# B&R Automation Studio project ProjectOrionBms (part 2)

#### AMS_Receive.st
```iecst
ACTION AMS_Receive:
	// Timer used for disconnection detection of AMS
	TON_amsDisconnected.PT   := T#200ms;	// Set timeout period
	TON_amsDisconnected.IN 	 := TRUE;		// Enable timer

	// Timer used for disconnection detection of shunt
	TON_shuntDisconnected.PT := T#200ms; 	// Set timeout period
	TON_shuntDisconnected.IN := TRUE;		// Enable timer

	FOR i := 0 TO 10 DO
		ArCanReceive_0(); // Run function block => Get next data frame

		(* If a new message has been received *)
		IF ArCanReceive_0.NewDataValid THEN
			messageCounterRec := messageCounterRec + 1;
			// Figure out if it is a shunt message
			IF ArCanReceive_0.ReceivedFrame.ID > SHUNT_ID_BASE AND ArCanReceive_0.ReceivedFrame.ID < (SHUNT_ID_BASE+16#30) THEN
				// Its a shunt message
				frameId := ArCanReceive_0.ReceivedFrame.ID - SHUNT_ID_BASE;
				// Look up message decoding
				CASE frameId OF
					16#021: msg_shunt_021;
					16#022: msg_shunt_022;
					16#023: msg_shunt_023;
//					16#025: msg_shunt_025;
					16#026: msg_shunt_026;
					16#027: msg_shunt_027;
					16#028: msg_shunt_028;
					ELSE (* Message not registered in system *)
				END_CASE

				(* Reset timer for disconnection detection *)
				TON_shuntDisconnected.IN := FALSE;

			// Figure out if the message is a ORION Message
			ELSIF ArCanReceive_0.ReceivedFrame.ID >= RX_ORION_ID_BASE AND ArCanReceive_0.ReceivedFrame.ID < (RX_ORION_ID_BASE+16#30) THEN
				// It is an ORION messagemm
				frameId := ArCanReceive_0.ReceivedFrame.ID - RX_ORION_ID_BASE;

				// Look up message decoding
				CASE frameId OF
					//16#000: msg_orion_000;
					16#001: msg_orion_001;
					16#002: msg_orion_002;
					16#003: msg_orion_003;
					16#004: msg_orion_004;
					16#010: msg_orion_010;
					16#011: msg_orion_011;

					ELSE // Not a message in the system
				END_CASE

			ELSE
				// Its an AMS message
				frameId := UDINT_TO_UINT(ArCanReceive_0.ReceivedFrame.ID) - RX_CAN_ID_BASE;

				// Look up message decoding
				CASE frameId OF
					16#000: msg_ams_000;
					16#011: msg_ams_011;
					16#012: msg_ams_012;
					16#013: msg_ams_013;
					16#014: msg_ams_014;
					ELSE (* Message not registered in system *)
				END_CASE

				TON_amsDisconnected.IN := FALSE; // Reset Timer
			END_IF;
		ELSE
			EXIT;
		END_IF
	END_FOR;

	(* If timeout occurres on AMS timer set AMS disconnect status flag *)
	TON_amsDisconnected();
	gAMS.status.disconnected := TON_amsDisconnected.Q;

	(* If timeout occurres on shunt timer set shunt disconnect status flag *)
	TON_shuntDisconnected();
	gShunt.status.disconnected := TON_shuntDisconnected.Q;

END_ACTION
```

### Program Logical/Dashboard/Dashboard

#### ErrorDashboard.st
```iecst
ACTION ErrorDashboard:

	gDashboard.outputs.com_error_Datalog 				:= NOT gDataLogging.status.dataloggingActive; // Datalogging not active
	gDashboard.outputs.com_error_SC 					:= NOT gSafetyChain.status.scOK_notEnabled; // Safety chain not ok
	gDashboard.outputs.com_error_Shunt 					:= NOT gShunt.status.ok; // Shunt error
	gDashboard.outputs.com_error_AMS 					:= NOT gAMS.status.ok; // AMS error
	gDashboard.outputs.com_error_Dashboard 				:= NOT gDashboard.status.ok; // Dashboard error
	gDashboard.outputs.com_error_3rd_Inv 				:= NOT gInverters.inverter[3].status.ok; // 3rd inverter error
	gDashboard.outputs.com_error_2nd_Inv 				:= NOT gInverters.inverter[2].status.ok; // 2nd inverter error
	gDashboard.outputs.com_error_1st_Inv 				:= NOT gInverters.inverter[1].status.ok; // 1st inverter error
	gDashboard.outputs.com_error_0_Inv 					:= NOT gInverters.inverter[0].status.ok; // [0] inverter error
	gDashboard.outputs.com_error_INS 					:= NOT gINS.status.ok; // INS error
	gDashboard.outputs.com_error_SteeringAngle 			:= gSteeringAngle.status.errorOutOfRange; // Steering angle out of range
	gDashboard.outputs.com_error_BreakPressure_Front 	:= gBraking.status.errorOutOfRangeFront; // Brake Pressure out-of-range (Front)
	gDashboard.outputs.com_error_BreakPressure_Back 	:= gBraking.status.errorOutOfRangeRear; // Brake Pressure out-of-range (Rear)
	gDashboard.outputs.com_error_TorquePedal 			:= gTorqueSensor.status.criticalError; // One of the Torque Pedal sensors out of range
	gDashboard.outputs.com_error_TorquePedal_Plausi 	:= gTorqueSensor.status.plausibilityError; // Plausibility error on Torque pedal
	gDashboard.outputs.com_error_RTDS 					:= NOT gRTDS.status.ok; // RTDS error
	gDashboard.outputs.com_error_Cooling	 			:= NOT gCooling.status.ok; // Cooling error
	gDashboard.outputs.com_error_LV 					:= gLowVoltageBattery.status.empty; // Low Voltage Battery critically low
	gDashboard.outputs.com_error_HighTemperature 		:= gCooling.status.warningHighTemperature;
END_ACTION
```

#### errors.st
```iecst
ACTION errors:
	// Change this variable to indicate what error is active in the system.
	// 0 = No error
	gDashboard.status.errorCode := 0;
END_ACTION
```

#### Main.st
```iecst
PROGRAM _INIT
	(* Device *)
	deviceName 						:= 'IF6.ST1.IF1';
	(* Bus *)
	ArCanSetBaudrate_0.Baudrate 	:= 1000000;
	(* Tramsit *)
	ArCanSend_0.Frame.Format 		:= arCAN_11BIT;
	(* Receive *)
	ArCanReceive_0.Format 			:= arCAN_11BIT;
	ArCanReceive_0.QueueSize		:= 100;
	ArCanReceive_0.IDMask			:= arCAN_RECEIVE_ALL;

	communicationState 				:= S_INIT;

	scLedState 						:= OFF;
	ledLVState 						:= 0;

	RX_CAN_ID_BASE 					:= 16#580;
	TX_CAN_ID_BASE 					:= 16#580;

END_PROGRAM

PROGRAM _CYCLIC

	(* Determine of the Dashboard has an error or is working properly*)
	gDashboard.status.ok := NOT gDashboard.status.DashboardDisconnected AND gDashboard.status.errorCode = 0;

	(* LED Control *)
	ledAMS;
	ledDV;
	ledEBS;
	ledIMD;
	ledLV;
	ledREADY;
	ledSC;
	ledTS_OFF;
	ErrorDashboard;

	(* Send and receive messages *)
	can;

	(* Error *)
	errors;

	// Log button presses
	IF EDGEPOS(gDashboard.inputs.di_button1) THEN
		gEventLog.newEventString := 'Button 1 pressed';
		logEvent;
	END_IF;
	IF EDGEPOS(gDashboard.inputs.di_button2) THEN
		gEventLog.newEventString := 'Button 2 pressed';
		logEvent;
	END_IF;
	IF EDGEPOS(gDashboard.inputs.di_button3) THEN
		gEventLog.newEventString := 'Button 3 pressed';
		logEvent;
	END_IF;
	IF EDGEPOS(gDashboard.inputs.di_button4) THEN
		gEventLog.newEventString := 'Button 4 pressed';
		logEvent;
	END_IF;
	IF EDGEPOS(gDashboard.inputs.di_buttonSafety) THEN
		gEventLog.newEventString := 'Button Safety pressed';
		logEvent;
	END_IF;
	IF EDGEPOS(gDashboard.inputs.di_buttonTractive) THEN
		gEventLog.newEventString := 'Button Tractive pressed';
		logEvent;
	END_IF;
	IF EDGEPOS(gDashboard.inputs.di_buttonDrive) THEN
		gEventLog.newEventString := 'Button Drive pressed';
		logEvent;
	END_IF;

END_PROGRAM

PROGRAM _EXIT

END_PROGRAM
```

#### ledTS_OFF.st
```iecst
(* Control the TS_OFF LED *)
ACTION ledTS_OFF:
	IF gStateMachine.status.state = STATE_INITIALIZE THEN
		gDashboard.outputs.do_ledTS_OFF := TRUE;
	ELSE
		gDashboard.outputs.do_ledTS_OFF := NOT (gStateMachine.status.state = STATE_TRACTIVE OR  gStateMachine.status.state = STATE_DRIVE);
	END_IF;

END_ACTION
```

#### Program Logical/Dashboard/Dashboard/Receive

##### Receive_Bus.st
```iecst
ACTION Receive_Bus:

	TON_disconnectTimer.PT := T#200ms;
	TON_disconnectTimer.IN := TRUE;

	FOR i := 0 TO UDINT_TO_USINT(LIMIT(0,ArCanReceive_0.QueueSize,255)) DO
		ArCanReceive_0(); // Run function block => Get next data frame
		(* If a new message has been received *)
		IF ArCanReceive_0.NewDataValid THEN
			(* Find which message is was and decode it *)

			frameIdOffset := ArCanReceive_0.ReceivedFrame.ID - RX_CAN_ID_BASE;
			CASE frameIdOffset OF
				16#050: msg_0x050;
				16#051: msg_0x051;
				16#052: msg_0x052;
				ELSE
				(* Message not registered in system *)
				gDashboard.status.unknownMessageReceived 	:= TRUE;
				gDashboard.status.unknownMessageID	 		:= ArCanReceive_0.ReceivedFrame.ID;
			END_CASE

			(* Enable timer to check if dashboard is disconnected *)
			TON_disconnectTimer.IN := FALSE;
			gDashboard.status.DashboardDisconnected := FALSE;
		ELSE
			EXIT;
		END_IF
	END_FOR;

	TON_disconnectTimer();

	(* If 200 ms is passed without message, set dashboard disconnect status flag *)
	IF TON_disconnectTimer.Q = TRUE THEN
		gDashboard.status.DashboardDisconnected := TRUE;
	END_IF

	gDashboard.status.canFramesLost := ArCanReceive_0.NumberOfLostFrames <> 0;

END_ACTION
```

### globalBraking.typ
```iecst
TYPE
	gBraking_cmd_typ : 	STRUCT
		brakePressureFront : INT;
		brakePressureRear : INT;
	END_STRUCT;
	gBraking_typ : 	STRUCT
		status : gBraking_status_typ;
		inputs : gBraking_inputs_typ;
		outputs : gBraking_outputs_typ;
		data : gBraking_data_typ;
		cmd : gBraking_cmd_typ;
	END_STRUCT;
	gBraking_status_typ : 	STRUCT
		ok : BOOL;
		errorOutOfRangeFront : BOOL;
		errorOutOfRangeRear : BOOL;
		softBraking : BOOL;
		hardBraking : BOOL;
	END_STRUCT;
	gBraking_inputs_typ : 	STRUCT
		ai_brakePressureFront : INT;
		ai_brakePressureRear : INT;
	END_STRUCT;
	gBraking_outputs_typ : 	STRUCT
		do_brakeLight : BOOL;
	END_STRUCT;
	gBraking_data_typ : 	STRUCT
		pressurePercentageFront : REAL;
		pressurePercentageRear : REAL;
		pressurePercentage : REAL;
		pressureBarRear : REAL;
		pressureBarFront : REAL;
	END_STRUCT;
END_TYPE
```

### globalBraking.var
```iecst
VAR
	gSoftBrakingForced : BOOL;
	gBraking : gBraking_typ;
END_VAR
```

### globalTorqueSensor.var
```iecst
VAR
	gTorqueSensor : gTorqueSensor_typ;
END_VAR
```

### Program Logical/Sensors/Sensors (IEC)

#### Main.st - Init, cyclic, exit code
```iecst
PROGRAM _INIT
	(* Initialize all the sensors *)
	// Accelerometer
	AccelerometerInit;

	// Braking Pedal Sensor
	BrakingPedalInit;

	// Torque Pedal Sensor
	TorquePedalInit;

	// Steering Angle Sensor
	SteeringAngleInit;

	// Low voltage battery
	LowVoltageBatteryInit;

	// Suspension Measurement
	SuspensionMeasInit;
END_PROGRAM

PROGRAM _CYCLIC
	//Accelerometer
	Accelerometer;

	// Handle Braking Pedal Sensor
	BrakingPedal;

	// Handle TorquePedal Sensor
	TorquePedal;

	// Handle Braking Pedal Sensor
	SteeringAngle;

	// Low voltage battery
	LowVoltageBattery;

	// Suspension Measurement
	SuspensionMeas;
END_PROGRAM

PROGRAM _EXIT
	(* Insert code here *)

END_PROGRAM
```

#### Types.typ - Local data types
```iecst
TYPE
	accelerometer_constants_typ : 	STRUCT
		VOLTAGE_MIN : UDINT;
		VOLTAGE_MAX : UDINT;
		MEASUREMENT_RES : UDINT;
		SENSOR_SUPPLY_VOLTAGE : UDINT;
		SENSITIVITY : REAL;
		ZERO_POINT : REAL;
	END_STRUCT;
	accelerometer_input_typ : 	STRUCT
		x_direction : INT;
		y_direction : INT;
		z_direction : INT;
	END_STRUCT;
	accelerometer_status_typ : 	STRUCT
		voltage_x : REAL;
		voltage_y : REAL;
		voltage_z : REAL;
		acceleration_x : REAL;
		acceleration_y : REAL;
		acceleration_z : REAL;
	END_STRUCT;
	accelerometer_typ : 	STRUCT
		constants : accelerometer_constants_typ;
		input : accelerometer_input_typ;
		status : accelerometer_status_typ;
	END_STRUCT;
	braking_pedal_constants_typ : 	STRUCT
		frontWarningLimitMaxMax : UINT;
		frontWarningLimitMax : UINT;
		frontWarningLimitMin : UINT;
		frontWarningLimitMinMin : UINT;
		rearWarningLimitMaxMax : UINT;
		rearWarningLimitMax : UINT;
		rearWarningLimitMin : UINT;
		rearWarningLimitMinMin : UINT;
		softBrakingLimit : UINT;
		hardBrakingLimit : UINT;
	END_STRUCT;
	braking_pedal_variables_typ : 	STRUCT
		brakingPedalFrontMax : UINT;
		brakingPedalFrontMin : UINT;
		brakingPedalRearMax : UINT;
		brakingPedalRearMin : UINT;
		slope : REAL;
	END_STRUCT;
	lv_battery_constants_typ : 	STRUCT
		HighLimit : REAL;
		LowLimit : REAL;
	END_STRUCT;
	lv_battery_variable_typ : 	STRUCT
		TON_batteryEmpty : TON;
		TON_batteryFull : TON;
	END_STRUCT;
	steering_angle_constants_typ : 	STRUCT
		highLimit : UINT;
		lowLimit : UINT;
		disconnectionLimit : UINT;
		MAX_ANGLE : REAL;
		MIN_ANGLE : REAL;
	END_STRUCT;
	steering_angle_variables_typ : 	STRUCT
		steeringWheelAngleStr : STRING[80];
		wheelAngleStr : STRING[80];
		leftValue : UINT;
		rightValue : UINT;
	END_STRUCT;
	suspension_const_typ : 	STRUCT
		VOLTAGE_MIN : UDINT;
		VOLTAGE_MAX : UDINT;
		MEASUREMENT_RES : UDINT;
		SENSOR_SUPPLY_VOLTAGE : UDINT;
		TRAVEL_RES : UDINT;
	END_STRUCT;
	suspension_input_typ : 	STRUCT
		linearPosSensor : ARRAY[0..3]OF INT;
	END_STRUCT;
	suspension_status_typ : 	STRUCT
		travelRR : REAL;
		travelFR : REAL;
		travelRL : REAL;
		travelFL : REAL;
		voltageRR : REAL;
		voltageFR : REAL;
		voltageRL : REAL;
		voltageFL : REAL;
	END_STRUCT;
	suspension_typ : 	STRUCT
		constants : suspension_const_typ;
		input : suspension_input_typ;
		status : suspension_status_typ;
	END_STRUCT;
	torque_pedal_constants_typ : 	STRUCT
		lowLimit2 : UINT;
		highLimit2 : UINT;
		lowLimit1 : UINT;
		highLimit1 : UINT;
		torqueOffUpperHysteresis : REAL;
		torqueOffLowerHysteresis : REAL;
	END_STRUCT;
	torque_pedal_variables_typ : 	STRUCT
		torquePedalMax2 : UINT;
		torquePedalMax1 : UINT;
		torquePedalMin2 : UINT;
		torquePedalMin1 : UINT;
		TON_torqueOff : TON;
		slope : REAL;
	END_STRUCT;
END_TYPE
```

#### Variables.var - Local variables
```iecst
VAR
	accelerometer : accelerometer_typ;
	brakingPedalVariables : braking_pedal_variables_typ;
	brakingPedalConstants : braking_pedal_constants_typ;
	torquePedalConstants : torque_pedal_constants_typ;
	torquePedalVariables : torque_pedal_variables_typ;
	steeringAngleConstants : steering_angle_constants_typ;
	steeringAngleVariables : steering_angle_variables_typ;
	lvBatteryConstants : lv_battery_constants_typ;
	lvBatteryVariables : lv_battery_variable_typ;
END_VAR
VAR RETAIN
	maxTorquePercentThrottle : USINT;
END_VAR
VAR
	suspension : suspension_typ;
END_VAR
```

#### BrakingPedal.st
```iecst
ACTION BrakingPedalInit:
	(* Sensor limit values *)
	brakingPedalVariables.brakingPedalRearMax 		:= 8000;
	brakingPedalVariables.brakingPedalRearMin 		:= 1655;
	brakingPedalVariables.brakingPedalFrontMax 		:= 8000;
	brakingPedalVariables.brakingPedalFrontMin 		:= 1655;

	(* Braking limits *)
	brakingPedalConstants.hardBrakingLimit			:= 5400;
	brakingPedalConstants.softBrakingLimit			:= 2200;

	(* Upper limit symboling an electrical fault *)
//	brakingPedalConstants.frontWarningLimitMaxMax 	:= brakingPedalVariables.brakingPedalFrontMax + 500;
//	brakingPedalConstants.rearWarningLimitMaxMax 	:= brakingPedalVariables.brakingPedalRearMax  + 500;
	brakingPedalConstants.frontWarningLimitMaxMax 	:= 15250;
	brakingPedalConstants.rearWarningLimitMaxMax 	:= 15250;

	(* Upper limit symboling a mechanical fault *)
	brakingPedalConstants.frontWarningLimitMax 		:= brakingPedalVariables.brakingPedalFrontMax + 100;
	brakingPedalConstants.rearWarningLimitMax 		:= brakingPedalVariables.brakingPedalRearMax  + 100;

	(* Lower limit symboling a mechanical fault *)
	brakingPedalConstants.frontWarningLimitMin 		:= brakingPedalVariables.brakingPedalFrontMin - 100;
	brakingPedalConstants.rearWarningLimitMin 		:= brakingPedalVariables.brakingPedalRearMin  - 100;

	(* Lower limit symboling an electrical fault *)
	brakingPedalConstants.frontWarningLimitMinMin 	:= brakingPedalVariables.brakingPedalFrontMin - 500;
	brakingPedalConstants.rearWarningLimitMinMin 	:= brakingPedalVariables.brakingPedalRearMin  - 500;

END_ACTION

ACTION BrakingPedal:
	(* Detect if brake pedal is being pressed lightly *)
	gBraking.status.softBraking 		 := INT_TO_UINT(gBraking.inputs.ai_brakePressureRear)  > brakingPedalConstants.softBrakingLimit OR
											gSoftBrakingForced;

	(* Detect hard braking *)
	gBraking.status.hardBraking 		 := INT_TO_UINT(gBraking.inputs.ai_brakePressureFront) > brakingPedalConstants.hardBrakingLimit OR
										    INT_TO_UINT(gBraking.inputs.ai_brakePressureRear)  > brakingPedalConstants.hardBrakingLimit;

	(* Control brakelight *)
	IF gStateMachine.status.state <> STATE_INITIALIZE THEN
		gBraking.outputs.do_brakeLight   := gBraking.status.softBraking;
	END_IF

	(* Check if brake pressures are out of range *)
	// If brake pressure front get above limit, an error message is shown.
	gBraking.status.errorOutOfRangeFront := INT_TO_UINT(gBraking.inputs.ai_brakePressureFront) >= brakingPedalConstants.frontWarningLimitMax OR
											INT_TO_UINT(gBraking.inputs.ai_brakePressureFront) <= brakingPedalConstants.frontWarningLimitMin;

	// If brake pressure rear get above limit, an error message is shown.
	gBraking.status.errorOutOfRangeRear := 	INT_TO_UINT(gBraking.inputs.ai_brakePressureRear) >= brakingPedalConstants.rearWarningLimitMax OR
											INT_TO_UINT(gBraking.inputs.ai_brakePressureRear) <= brakingPedalConstants.rearWarningLimitMin;

	(* Calculate pedal percentages *)
	IF NOT gBraking.status.errorOutOfRangeFront THEN
		brakingPedalVariables.slope := (100.00)/(UINT_TO_REAL(brakingPedalVariables.brakingPedalFrontMax) - UINT_TO_REAL(brakingPedalVariables.brakingPedalFrontMin));
		gBraking.data.pressurePercentageFront := LIMIT(0 ,brakingPedalVariables.slope * (INT_TO_REAL(gBraking.inputs.ai_brakePressureFront)-UINT_TO_REAL(brakingPedalVariables.brakingPedalFrontMin)),100);
	ELSE
		gBraking.data.pressurePercentageFront := 0;
	END_IF;

	IF NOT gBraking.status.errorOutOfRangeRear THEN
		brakingPedalVariables.slope := (100.00)/(UINT_TO_REAL(brakingPedalVariables.brakingPedalRearMax) - UINT_TO_REAL(brakingPedalVariables.brakingPedalRearMin));
		gBraking.data.pressurePercentageRear := LIMIT(0 ,brakingPedalVariables.slope * (INT_TO_REAL(gBraking.inputs.ai_brakePressureRear)-UINT_TO_REAL(brakingPedalVariables.brakingPedalRearMin)),100);
	ELSE
		gBraking.data.pressurePercentageRear := 0;
	END_IF;

	gBraking.data.pressurePercentage := (gBraking.data.pressurePercentageFront + gBraking.data.pressurePercentageRear)/2.0;

	(* Determine if the brake pedal + sensors are working properly *)
	gBraking.status.ok := NOT gBraking.status.errorOutOfRangeFront AND NOT gBraking.status.errorOutOfRangeRear;

	// Calculate actual pressure
	gBraking.data.pressureBarFront 	:= ((INT_TO_REAL(gBraking.inputs.ai_brakePressureFront)*10/32768)-0.5)*40;
	gBraking.data.pressureBarRear	:= ((INT_TO_REAL(gBraking.inputs.ai_brakePressureRear)*10/32768)-0.5)*40;

END_ACTION
```

#### TorquePedal.st
```iecst
ACTION TorquePedalInit:
	(* Sensor edge values *)
	torquePedalVariables.torquePedalMin1 	:= 13636;
	torquePedalVariables.torquePedalMin2 	:= 2415;
	torquePedalVariables.torquePedalMax1 	:= 21181;
	torquePedalVariables.torquePedalMax2 	:= 7947;

	// Constant for limit torque percent
	IF maxTorquePercentThrottle = 0 THEN
		maxTorquePercentThrottle := 50; // Change to 100 for max torque, 50 is a bit over nominal  torque. Max= 21NM, Nominal = 9,8Nm
	END_IF;
	gTorqueSensor.status.maxTorquePercent := maxTorquePercentThrottle;

	(* Range for torque sensor 1 *)
	torquePedalConstants.highLimit1 := torquePedalVariables.torquePedalMax1 + 200;
	torquePedalConstants.lowLimit1  := 0;

	(* Range for torque sensor 2 *)
	torquePedalConstants.highLimit2 := torquePedalVariables.torquePedalMax2 + 200;
	torquePedalConstants.lowLimit2 	:= 0;

	(* Torque off hysteresis values *)
	torquePedalConstants.torqueOffUpperHysteresis := 25; // [%]
	torquePedalConstants.torqueOffLowerHysteresis := 5;  // [%]

	(* Plausibility check disable (for test setup) *)
	gTorqueSensor.cmd.disablePlausibilityCheck := FALSE;
END_ACTION

ACTION TorquePedal:
	// Percent of MAX torque at full throttle:
	gTorqueSensor.status.maxTorquePercent := maxTorquePercentThrottle;

	gTorqueSensor.status.errorOutOfRangeSensor1 := 	INT_TO_UINT(gTorqueSensor.inputs.torque1) > torquePedalConstants.highLimit1 OR
													INT_TO_UINT(gTorqueSensor.inputs.torque1) < torquePedalConstants.lowLimit1;

	gTorqueSensor.status.errorOutOfRangeSensor2 := 	INT_TO_UINT(gTorqueSensor.inputs.torque2) > torquePedalConstants.highLimit2 OR
													INT_TO_UINT(gTorqueSensor.inputs.torque2) < torquePedalConstants.lowLimit2;

	(* Calculate pedal percentages *)

	// Sensor 1
	IF NOT gTorqueSensor.status.errorOutOfRangeSensor1 THEN
		torquePedalVariables.slope := (100)/(UINT_TO_REAL(torquePedalVariables.torquePedalMax1) - UINT_TO_REAL(torquePedalVariables.torquePedalMin1));
		gTorqueSensor.data.torque1Percent := LIMIT(0 ,torquePedalVariables.slope * (INT_TO_REAL(gTorqueSensor.inputs.torque1)-(10+UINT_TO_REAL(torquePedalVariables.torquePedalMin1))),100);
	ELSE
		gTorqueSensor.data.torque1Percent := 0;
	END_IF;
	// gTorqueSensor.status.maxTorquePercent TODO: USE THIS FOR SCALING
	// Sensor 2
	IF NOT gTorqueSensor.status.errorOutOfRangeSensor2 THEN
		torquePedalVariables.slope := (100)/(UINT_TO_REAL(torquePedalVariables.torquePedalMax2) - UINT_TO_REAL(torquePedalVariables.torquePedalMin2));
		gTorqueSensor.data.torque2Percent := LIMIT(0 ,torquePedalVariables.slope * (INT_TO_REAL(gTorqueSensor.inputs.torque2)-UINT_TO_REAL(torquePedalVariables.torquePedalMin2)),100);
	ELSE
		gTorqueSensor.data.torque2Percent := 0;
	END_IF;

	// Sensor 1 is arbitrarily taken to be the torque percentage
	// Value is then scaled by desired power
	gTorqueSensor.status.torquePercentage := gTorqueSensor.data.torque1Percent*gTorqueSensor.status.maxTorquePercent/100;

	(* Test if torque sensor values are out of range of each other*)
	TorqueSensorsOutOfRange;
	TorqueOff;

	(* Report critical error if either of the torque pedal sensors leave their working range *)
	gTorqueSensor.status.criticalError := gTorqueSensor.status.errorOutOfRangeSensor1 OR gTorqueSensor.status.errorOutOfRangeSensor2 OR gTorqueSensor.status.plausibilityError;

	(* Determine if the torque pedal is working properly *)
	gTorqueSensor.status.ok := NOT gTorqueSensor.status.criticalError;

END_ACTION

(* Test if torque pedals are more than 10% different than each other *)
ACTION TorqueSensorsOutOfRange:
	IF gTorqueSensor.cmd.disablePlausibilityCheck THEN
		gTorqueSensor.status.plausibilityError := FALSE;
	ELSE
		// check if torque sensor 1 and 2 vary more than 5 %
		gTorqueSensor.status.plausibilityError := ABS(gTorqueSensor.data.torque1Percent - gTorqueSensor.data.torque2Percent) > 5;
	END_IF;
END_ACTION

ACTION TorqueOff:
	IF gTorqueSensor.status.torqueEnabled THEN
		(* Test the criterias for turning off the torque. If they are met start timer *)
		IF 	gBraking.status.softBraking AND
			(gTorqueSensor.data.torque1Percent >= torquePedalConstants.torqueOffUpperHysteresis OR
			 gTorqueSensor.data.torque2Percent >= torquePedalConstants.torqueOffUpperHysteresis OR
		 	 gORION.data.packPower >= 5.0) THEN

			torquePedalVariables.TON_torqueOff.PT := T#250ms;	// Set timer duration TODO: Change to 500 that is the limit in the rules
			torquePedalVariables.TON_torqueOff.IN := TRUE;		// Start timer
		ELSE
			torquePedalVariables.TON_torqueOff.IN := FALSE;		// Else stop timer
		END_IF

		IF torquePedalVariables.TON_torqueOff.Q THEN			// If timer runs out
			gTorqueSensor.status.torqueEnabled := FALSE;		// Remove torque
		ELSE
			gTorqueSensor.status.torqueEnabled := TRUE;			// Else keep torque
		END_IF;
	ELSE
		(* Test the criterias for turning on the torque *)
		gTorqueSensor.status.torqueEnabled := 	gTorqueSensor.data.torque1Percent < torquePedalConstants.torqueOffLowerHysteresis AND
												gTorqueSensor.data.torque2Percent < torquePedalConstants.torqueOffLowerHysteresis AND (NOT gBraking.status.softBraking);
		torquePedalVariables.TON_torqueOff.IN := FALSE;			// Make sure the torque timer is stopped
	END_IF
	torquePedalVariables.TON_torqueOff();						// Run torque timer
END_ACTION
```

#### SteeringAngle.st
```iecst
ACTION SteeringAngleInit:
	(* Sensor limit values *)
	steeringAngleVariables.leftValue 	:= 7460;
	steeringAngleVariables.rightValue 	:= 25580;

	(* Error detection values *)
	steeringAngleConstants.disconnectionLimit := 300;
	steeringAngleConstants.lowLimit 	:= steeringAngleVariables.leftValue  - 500;
	steeringAngleConstants.highLimit 	:= steeringAngleVariables.rightValue + 500;

	steeringAngleConstants.MAX_ANGLE 	:=  100.00;
	steeringAngleConstants.MIN_ANGLE 	:= -100.00;
END_ACTION

ACTION SteeringAngle:
	(* 	Check if sensor input is within working range
		If not report an error  	*)
	gSteeringAngle.status.disconnected := INT_TO_UINT(gSteeringAngle.inputs.angleSensor) < steeringAngleConstants.disconnectionLimit;
	gSteeringAngle.status.errorOutOfRange := (NOT gSteeringAngle.status.disconnected) AND (INT_TO_UINT(gSteeringAngle.inputs.angleSensor) > steeringAngleConstants.highLimit OR INT_TO_UINT(gSteeringAngle.inputs.angleSensor) < steeringAngleConstants.lowLimit);
	(* Summerize errors *)
	gSteeringAngle.status.error := gSteeringAngle.status.disconnected OR gSteeringAngle.status.errorOutOfRange;

	(* Calculate steering angle *)
	IF NOT gSteeringAngle.status.error THEN
		// No error
		IF INT_TO_UINT(gSteeringAngle.inputs.angleSensor) < steeringAngleVariables.leftValue THEN
			gSteeringAngle.data.angleDegrees := steeringAngleConstants.MAX_ANGLE;
		ELSIF INT_TO_UINT(gSteeringAngle.inputs.angleSensor) > steeringAngleVariables.rightValue THEN
			gSteeringAngle.data.angleDegrees := steeringAngleConstants.MIN_ANGLE;
		ELSE
			gSteeringAngle.data.angleDegrees := LIMIT(-100, (INT_TO_REAL(gSteeringAngle.inputs.angleSensor) - UINT_TO_REAL(steeringAngleVariables.leftValue))/(UINT_TO_REAL(steeringAngleVariables.rightValue) - UINT_TO_REAL(steeringAngleVariables.leftValue)) *
			(ABS(steeringAngleConstants.MAX_ANGLE) + ABS(steeringAngleConstants.MIN_ANGLE)) + steeringAngleConstants.MIN_ANGLE, 100)*(-1);
		END_IF;
	ELSE
		// Error
		gSteeringAngle.data.angleDegrees := 0;
	END_IF

	(* Determine if the steering angle sensor is working properly *)
	gSteeringAngle.status.ok := NOT gSteeringAngle.status.disconnected AND NOT gSteeringAngle.status.error;

	// Visualization action
	hmi;

END_ACTION
```

#### hmi.st
```iecst
ACTION hmi:

	(* Wheels *)
	gSteeringAngle.data.wheelAngle := gSteeringAngle.data.angleDegrees / 3.33;
	gSteeringAngle.status.wheelSVG := '[{"select":"#wheel","duration":0,"spin":[';
	steeringAngleVariables.wheelAngleStr := REAL_TO_STRING(gSteeringAngle.data.wheelAngle);
	brdkStrCat(ADR(gSteeringAngle.status.wheelSVG), ADR(steeringAngleVariables.wheelAngleStr));
	brdkStrCat(ADR(gSteeringAngle.status.wheelSVG), ADR(',55,85]}]'));

	(* Steering angle transformation and show if buttons are pressed*)
	gSteeringAngle.status.steeringWheelSVG := '[';
	steeringAngleVariables.steeringWheelAngleStr := REAL_TO_STRING(gSteeringAngle.data.angleDegrees);
	brdkStrCat(ADR(gSteeringAngle.status.steeringWheelSVG),ADR('{"select":"#all","duration":0,"spin":['));
	brdkStrCat(ADR(gSteeringAngle.status.steeringWheelSVG),ADR(steeringAngleVariables.steeringWheelAngleStr));
	brdkStrCat(ADR(gSteeringAngle.status.steeringWheelSVG),ADR(',290,245]}'));

	brdkStrCat(ADR(gSteeringAngle.status.steeringWheelSVG),ADR(']'));
END_ACTION
```

#### SuspensionMeas.st
```iecst
ACTION SuspensionMeasInit:
	suspension.constants.VOLTAGE_MIN 			:= 0;
	suspension.constants.VOLTAGE_MAX 			:= 32;
	suspension.constants.MEASUREMENT_RES		:= 32767;
	suspension.constants.SENSOR_SUPPLY_VOLTAGE 	:= 24;
	suspension.constants.TRAVEL_RES				:= 50; // [mm]
END_ACTION

ACTION SuspensionMeas:
	// Some calculation of the suspension travel in mm, based on analog voltage reading.
	suspension.status.voltageFL := UDINT_TO_REAL((suspension.constants.VOLTAGE_MAX - suspension.constants.VOLTAGE_MIN) * suspension.input.linearPosSensor[0]) / suspension.constants.MEASUREMENT_RES;
	suspension.status.travelFL 	:= suspension.status.voltageFL/suspension.constants.SENSOR_SUPPLY_VOLTAGE * suspension.constants.TRAVEL_RES;

	// Some calculation of the suspension travel in mm, based on analog voltage reading.
	suspension.status.voltageRL := UDINT_TO_REAL((suspension.constants.VOLTAGE_MAX - suspension.constants.VOLTAGE_MIN) * suspension.input.linearPosSensor[1]) / suspension.constants.MEASUREMENT_RES;
	suspension.status.travelRL 	:= suspension.status.voltageRL/suspension.constants.SENSOR_SUPPLY_VOLTAGE * suspension.constants.TRAVEL_RES;

	// Some calculation of the suspension travel in mm, based on analog voltage reading.
	suspension.status.voltageFR := UDINT_TO_REAL((suspension.constants.VOLTAGE_MAX - suspension.constants.VOLTAGE_MIN) * suspension.input.linearPosSensor[2]) / suspension.constants.MEASUREMENT_RES;
	suspension.status.travelFR 	:= suspension.status.voltageFR/suspension.constants.SENSOR_SUPPLY_VOLTAGE * suspension.constants.TRAVEL_RES;

	// Some calculation of the suspension travel in mm, based on analog voltage reading.
	suspension.status.voltageRR := UDINT_TO_REAL((suspension.constants.VOLTAGE_MAX - suspension.constants.VOLTAGE_MIN) * suspension.input.linearPosSensor[3]) / suspension.constants.MEASUREMENT_RES;
	suspension.status.travelRR	:= suspension.status.voltageRR/suspension.constants.SENSOR_SUPPLY_VOLTAGE * suspension.constants.TRAVEL_RES;
END_ACTION
```

#### Accelerometer.st
```iecst
ACTION AccelerometerInit:
	accelerometer.constants.VOLTAGE_MIN 			:= 0;
	accelerometer.constants.VOLTAGE_MAX 			:= 10;
	accelerometer.constants.MEASUREMENT_RES		    := 32767;
	accelerometer.constants.SENSOR_SUPPLY_VOLTAGE 	:= 3;
	accelerometer.constants.SENSITIVITY				:= 0.3;
	accelerometer.constants.ZERO_POINT				:= 1.5;
END_ACTION

ACTION Accelerometer:

	// Some calculation of the acceleration in g, based on analog voltage reading.
	accelerometer.status.voltage_x := UDINT_TO_REAL((accelerometer.constants.VOLTAGE_MAX - accelerometer.constants.VOLTAGE_MIN) * accelerometer.input.x_direction) / accelerometer.constants.MEASUREMENT_RES;
	accelerometer.status.acceleration_x := (accelerometer.status.voltage_x - accelerometer.constants.ZERO_POINT) / accelerometer.constants.SENSITIVITY;

	// Some calculation of the acceleration in g, based on analog voltage reading.
	accelerometer.status.voltage_y := UDINT_TO_REAL((accelerometer.constants.VOLTAGE_MAX - accelerometer.constants.VOLTAGE_MIN) * accelerometer.input.y_direction) / accelerometer.constants.MEASUREMENT_RES;
	accelerometer.status.acceleration_y := (accelerometer.status.voltage_y - accelerometer.constants.ZERO_POINT) / accelerometer.constants.SENSITIVITY;

	// Some calculation of the acceleration in g, based on analog voltage reading.
	accelerometer.status.voltage_z := UDINT_TO_REAL((accelerometer.constants.VOLTAGE_MAX - accelerometer.constants.VOLTAGE_MIN) * accelerometer.input.z_direction) / accelerometer.constants.MEASUREMENT_RES;
	accelerometer.status.acceleration_z := (accelerometer.status.voltage_z - accelerometer.constants.ZERO_POINT) / accelerometer.constants.SENSITIVITY;

END_ACTION
```

### globalSensorNet.typ
```iecst
TYPE
	gSensorNet_typ : 	STRUCT
		status : gSensorNet_status_typ;
		inputs : gSensorNet_inputs_typ;
		outputs : gSensorNet_outputs_typ;
		cmd : gSensorNet_cmd_typ;
		data : gSensorNet_data_typ;
	END_STRUCT;
	gSensorNet_status_typ : 	STRUCT
		dummy : USINT;
	END_STRUCT;
	gSensorNet_data_typ : 	STRUCT
		coolingTemp1 : sensorNetVariable_typ;
	END_STRUCT;
	gSensorNet_inputs_typ : 	STRUCT
		dummy : USINT;
	END_STRUCT;
	gSensorNet_cmd_typ : 	STRUCT
		dummy : USINT;
	END_STRUCT;
	gSensorNet_outputs_typ : 	STRUCT
		dummy : USINT;
	END_STRUCT;
	sensorNetVariable_typ : 	STRUCT
		input : INT;
		polyCoeffs : ARRAY[0..SENSOR_NET_POLY_LEN]OF REAL;
		value : REAL;
	END_STRUCT;
END_TYPE
```

### Program Logical/SensorNet/globalSensorNet (IEC)

#### Main.st - Init, cyclic, exit code
```iecst
PROGRAM _INIT
	(* Device *)
	deviceName 						:= 'IF6.ST1.IF2';
	(* Bus *)
	ArCanSetBaudrate_0.Baudrate 	:= 1000000;
	(* Tramsit *)
	ArCanSend_0.Frame.Format 		:= arCAN_11BIT;
	(* Receive *)
	ArCanReceive_0.Format 			:= arCAN_11BIT;
	ArCanReceive_0.QueueSize		:= 100;
	ArCanReceive_0.IDMask			:= arCAN_RECEIVE_ALL;

	communicationState 				:= S_INIT;

	RX_CAN_ID_BASE 					:= 16#600;
	TX_CAN_ID_BASE 					:= 16#600;

END_PROGRAM

PROGRAM _CYCLIC

	(* Send and receive messages *)
	can;

	calculateSensorNetOut_0(input := gSensorNet.data.coolingTemp1.input, polyCoeffs := gSensorNet.data.coolingTemp1.polyCoeffs);
	gSensorNet.data.coolingTemp1.value := calculateSensorNetOut_0.output;

END_PROGRAM

PROGRAM _EXIT
	(* Insert code here *)

END_PROGRAM
```

#### Variables.var - Local variables
```iecst
VAR
	a : ARRAY[0..SENSOR_NET_POLY_LEN] OF REAL;
	i : USINT;
	y : REAL;
	x : INT;
	deviceName : STRING[127];
	calculateSensorNetOut_0 : calculateSensorNetOut;
	ArCanSetBaudrate_0 : ArCanSetBaudrate;
	communicationState : CAN_STATES;
	ArCanSend_0 : ArCanSend;
	ArCanReceive_0 : ArCanReceive;
	TON_sendTimer : TON;
	TON_disconnectTimer : TON;
END_VAR
```

#### can.st
```iecst
ACTION can:

	CASE communicationState OF
		S_INIT:	// Init
			(* PLC is not simulated. It is run on an actual PLC *)
			IF NOT gIsSimulation THEN

				(* Configure CAN port *)
				ArCanSetBaudrate_0.DeviceName	:= deviceName;

				ArCanSetBaudrate_0.Execute 	:= TRUE;
				IF ArCanSetBaudrate_0.Done THEN
					communicationState 	:= S_INIT_TX;
				END_IF;

				IF ArCanSetBaudrate_0.Error THEN
					communicationState 	:= S_ERROR;
				END_IF;

			ELSE
				(* PLC is simulated. It is run in the simulator and no hardware is connnected *)
				communicationState 		:= S_IDLE;
			END_IF;

		S_INIT_TX:	// Init Transmit
			(* Configure send function block *)
			ArCanSend_0.Enable 			:= TRUE;
			ArCanSend_0.DeviceName 		:= deviceName;

			IF ArCanSend_0.Active THEN
				communicationState 		:= S_INIT_RX;
			END_IF;

			IF ArCanSend_0.Error THEN
				communicationState 		:= S_ERROR;
			END_IF;

		S_INIT_RX:	// Init Receive
			(* Configure receive function block *)
			ArCanReceive_0.Enable 			:= TRUE;
			ArCanReceive_0.DeviceName 		:= deviceName;

			IF ArCanReceive_0.Active THEN
				(* CAN port successfully enabled *)
				communicationState 		:= S_RUNNING;
			END_IF;

			IF ArCanReceive_0.Error THEN
				communicationState 		:= S_ERROR;
			END_IF

		S_RUNNING:	// Running
			Send_Bus;		// Handle transmit
			Receive_Bus;	// Handle receive

		S_ERROR: // Error
			IF ArCanSend_0.Error THEN
				ArCanSend_0(Enable := FALSE);
				ArCanSend_0(Enable := TRUE);
			END_IF;

			IF ArCanReceive_0.Error THEN
				ArCanReceive_0(Enable := FALSE);
				ArCanReceive_0(Enable := TRUE);
			END_IF;

			IF ArCanReceive_0.Error = FALSE AND ArCanSend_0.Error = FALSE AND ArCanSetBaudrate_0.Error = FALSE THEN
				communicationState 		:= S_INIT;
			END_IF;
		S_IDLE: // Do nothing
	END_CASE

	IF NOT gIsSimulation THEN
		ArCanSetBaudrate_0();
		ArCanSend_0();
		ArCanReceive_0();
	END_IF;

END_ACTION
```

#### Receive_Bus.st
```iecst
ACTION Receive_Bus:
	// Timer used for disconnection detection of Sensor Network
	TON_disconnectTimer.PT   := T#200ms;	// Set timeout period
	TON_disconnectTimer.IN 	 := TRUE;		// Enable timer

	FOR i := 0 TO UDINT_TO_USINT(LIMIT(0,ArCanReceive_0.QueueSize,255)) DO
		ArCanReceive_0(); // Run function block => Get next data frame

		(* If a new message has been received *)
		IF ArCanReceive_0.NewDataValid THEN
			(* Find which message is was and decode it *)

			frameIdOffset := ArCanReceive_0.ReceivedFrame.ID - RX_CAN_ID_BASE;
			// Look up message decoding
			CASE frameIdOffset OF
//				16#050: msg_0x050;	Setup messages
//				16#051: msg_0x051;	Setup messages
//				16#052: msg_0x052;	Setup messages
				ELSE
				(* Message not registered in system *)
			END_CASE

			(* Enable timer to check if Sensor Network is disconnected *)
			TON_disconnectTimer.IN := FALSE;
		ELSE
			EXIT;
		END_IF
	END_FOR;

	TON_disconnectTimer();

	(* If 200 ms is passed without message, set dashboard disconnect status flag *)
	IF TON_disconnectTimer.Q = TRUE THEN
		gDashboard.status.DashboardDisconnected := TRUE;
	END_IF

END_ACTION
```

#### receive_messages.st
```iecst
ACTION msg_0x050:

END_ACTION

ACTION msg_0x051:

END_ACTION

ACTION msg_0x052:

END_ACTION
```

#### Send_Bus.st
```iecst
ACTION Send_Bus:
	(* Set timer *)
	TON_sendTimer.PT := T#100ms;

	(* If timer runs out *)
	IF NOT gIsSimulation THEN
		IF TON_sendTimer.Q THEN
			CASE msgIndex OF
				//	0: msg_0x000; 	Make messages
				//	1: msg_0x001;	Make messages
				//	2: msg_0x002;	Make messages
				ELSE
				END_CASE;
			ArCanSend_0(SendFrame := TRUE);
			ArCanSend_0(SendFrame := FALSE);

			msgIndex := msgIndex + 1;
			IF msgIndex > 2 THEN
				msgIndex := 0;
			END_IF;

			(* Reset timer *)
			TON_sendTimer(IN:=FALSE);
		END_IF;

	END_IF;

	(* Start timer *)
	TON_sendTimer(IN:=TRUE);

	ArCanSend_0();
END_ACTION
```

#### send_messages.st
```iecst
ACTION msg_0x000:
	ArCanSend_0.Frame.ID 		  := TX_CAN_ID_BASE + 16#000; // CAN-ID
	ArCanSend_0.Frame.DataLength  := 6; 	 // Datalength

	speed 			:=	REAL_TO_INT(  gINS.data.actLonVelocity_kmh * 10.00 );
	soc 			:=	REAL_TO_INT(  gAMS.data.stateOfCharge * 10.00 );
	maxTemperature  := 	REAL_TO_UINT(MAX(gInverters.inverter[0].data.tempMotor, gInverters.inverter[1].data.tempMotor, gInverters.inverter[2].data.tempMotor, gInverters.inverter[3].data.tempMotor) * 10.00);

	memcpy(ADR(ArCanSend_0.Frame.Data[0]), ADR( speed 			), 2);
	memcpy(ADR(ArCanSend_0.Frame.Data[2]), ADR( soc 			), 2);
	memcpy(ADR(ArCanSend_0.Frame.Data[4]), ADR( maxTemperature	), 2);

END_ACTION

ACTION msg_0x001:

END_ACTION

ACTION msg_0x002:

END_ACTION

ACTION msg_0x003:

END_ACTION
```

### globalRTDS.typ
```iecst
TYPE
	gRTDS_typ : 	STRUCT
		status : gRTDS_status_typ;
		inputs : gRTDS_inputs_typ;
		outputs : gRTDS_outputs_typ;
		cmd : gRTDS_cmd_typ;
		data : gRTDS_data_typ;
	END_STRUCT;
	gRTDS_status_typ : 	STRUCT
		ok : BOOL;
		RTDS_Off : BOOL;
		RTDS_Disconnected : BOOL;
		RTDS_On : BOOL;
	END_STRUCT;
	gRTDS_data_typ : 	STRUCT
		dummy : USINT;
	END_STRUCT;
	gRTDS_inputs_typ : 	STRUCT
		im_RTDS_Current : INT;
	END_STRUCT;
	gRTDS_cmd_typ : 	STRUCT
		en_RTDS : BOOL;
	END_STRUCT;
	gRTDS_outputs_typ : 	STRUCT
		do_RTDS : BOOL;
	END_STRUCT;
END_TYPE
```

### Program Logical/Actuators/Output/RTDS

#### RTDS.st
```iecst
ACTION RtdsInit:
	rtdsConstants.RTDSCurrent := 55;
	rtdsVariables.TON_RTDS.PT := T#2s;
END_ACTION

ACTION Rtds:
	// Check if RTDS is turned on.
	gRTDS.status.RTDS_On  := gRTDS.outputs.do_RTDS AND gRTDS.inputs.im_RTDS_Current > rtdsConstants.RTDSCurrent;
	gRTDS.status.RTDS_Off := NOT gRTDS.status.RTDS_On;

	(* Check if the RTDS should be on and compare it with the current, and set a status flag *)
	gRTDS.status.RTDS_Disconnected := gRTDS.outputs.do_RTDS AND gRTDS.inputs.im_RTDS_Current < rtdsConstants.RTDSCurrent;

	// If the car is switched into state DRIVE, start RTDS
	IF gStateMachine.status.state = STATE_DRIVE AND gStateMachine.status.stateOld <> STATE_DRIVE AND NOT gRTDS.cmd.en_RTDS THEN
		gRTDS.cmd.en_RTDS := TRUE;		(* Set command RTDS = true *)
	END_IF;

	// Check for command to turn on timer
	IF gRTDS.cmd.en_RTDS THEN
		rtdsVariables.TON_RTDS.IN 	:= TRUE; (* Enable timer *)
		gRTDS.outputs.do_RTDS 		:= TRUE; (* Set output high *)
	END_IF

	rtdsVariables.TON_RTDS();			(* Handle timer *)

	// If timer runs out
	IF rtdsVariables.TON_RTDS.Q THEN
		gRTDS.cmd.en_RTDS 			:= FALSE; (* Disable command *)
		gRTDS.outputs.do_RTDS 		:= FALSE; (* Set output low *)
		rtdsVariables.TON_RTDS.IN 	:= FALSE; (* Disable timer *)
	END_IF

	(* Determine if the RTDS is working properly *)
	gRTDS.status.ok := NOT gRTDS.status.RTDS_Disconnected;

END_ACTION
```

### globalCooling.typ
```iecst
TYPE
	gCooling_typ : 	STRUCT
		outputs : gCooling_outputs_typ;
		inputs : gCooling_inputs_typ;
		data : gCooling_data_typ;
		cmd : gCooling_cmd_typ;
		status : gCooling_status_typ;
	END_STRUCT;
	gCooling_outputs_typ : 	STRUCT
		do_fan : ARRAY[0..NUMBER_OF_FANS]OF BOOL;
		do_pump : ARRAY[0..NUMBER_OF_PUMPS]OF BOOL;
	END_STRUCT;
	gCooling_inputs_typ : 	STRUCT
		ai_coolingTemp : ARRAY[0..NUMBER_OF_COOLING_SENSORS]OF INT;
		im_pumpCurrent : ARRAY[0..NUMBER_OF_PUMPS]OF INT;
	END_STRUCT;
	gCooling_cmd_typ : 	STRUCT
		manualMode : BOOL;
		inverterMaxTemp : REAL;
		motorMaxTemp : REAL;
		motorTempStartPump : REAL;
		inverterTempStartPump : REAL;
	END_STRUCT;
	gCooling_status_typ : 	STRUCT
		ok : BOOL;
		error : BOOL;
		pumpError : ARRAY[0..1]OF BOOL;
		pumpState : ARRAY[0..1]OF PUMP_STATES;
		warningHighTemperature : BOOL;
		warningInverterHighTemp : BOOL;
		warningMotorHighTemp : BOOL;
	END_STRUCT;
	gCooling_data_typ : 	STRUCT
		coolingSysTemp : ARRAY[0..NUMBER_OF_COOLING_SENSORS]OF REAL;
	END_STRUCT;
	PUMP_STATES :
		(
		PUMP_STATE_OK,
		PUMP_STATE_NO_WATER,
		PUMP_STATE_NOT_CONNECTED
		);
END_TYPE
```

### Program Logical/CoolingSystem/COOLING

#### Variables.var
```iecst
VAR
	inverterMaxTemp : REAL;
	motorMaxTemp : REAL;
	COOLING_MODE_STATE : USINT := 0;
	pumpOffCurrent : UINT;
	pumpOnCurrent : UINT;
	i : USINT;
END_VAR
```

#### Main.st
```iecst
PROGRAM _INIT
	pumpOffCurrent := 1000;
	pumpOnCurrent  := 9500;
	gCooling.cmd.manualMode := FALSE;
	//gCooling.outputs.do_pump[1] := TRUE;
	FOR i := 0 TO 1 DO
		gCooling.outputs.do_pump[i] 	:= TRUE;
		gCooling.outputs.do_fan[i] 		:= TRUE;
		//gCooling.outputs.do_pump[i] 	:= FALSE;
		//gCooling.outputs.do_fan[i] 		:= FALSE;
	END_FOR

	gCooling.status.warningHighTemperature := FALSE;

	gCooling.cmd.inverterMaxTemp 	:= 60.0;
	gCooling.cmd.motorMaxTemp 		:= 100.0;

	gCooling.cmd.motorTempStartPump := 30;
	gCooling.cmd.inverterTempStartPump := 35;

END_PROGRAM

PROGRAM _CYCLIC

	motorMaxTemp := MAX(gInverters.inverter[0].data.tempMotor   , gInverters.inverter[1].data.tempMotor,    gInverters.inverter[2].data.tempMotor,    gInverters.inverter[3].data.tempMotor);
	inverterMaxTemp := MAX(gInverters.inverter[0].data.tempInverter, gInverters.inverter[1].data.tempInverter, gInverters.inverter[2].data.tempInverter, gInverters.inverter[3].data.tempInverter);

	CASE COOLING_MODE_STATE OF
		0: // AUTO MODE
			IF gDashboard.inputs.di_button2 AND (gInverters.inverter[0].data.actualVelocityKmh < 1) THEN
				COOLING_MODE_STATE := 10;
			END_IF;
//			IF gStateMachine.status.state = STATE_DRIVE THEN
//				COOLING_MODE_STATE := 10;
//			END_IF;
		10: // going to MANUAL MODE
			IF NOT gDashboard.inputs.di_button2 THEN
				gCooling.cmd.manualMode := TRUE;
				gCooling.outputs.do_pump[1] := TRUE;
				COOLING_MODE_STATE := 20;
			END_IF;

		20: // MANUAL MODE
			IF gDashboard.inputs.di_button2 AND (gInverters.inverter[0].data.actualVelocityKmh < 1) THEN
				COOLING_MODE_STATE := 30;
			END_IF;

		30: // going to  auto mode
			IF NOT gDashboard.inputs.di_button2 THEN
				gCooling.cmd.manualMode := FALSE;
				gCooling.outputs.do_pump[1] := FALSE;
				COOLING_MODE_STATE := 0;
			END_IF
	END_CASE;

	// If the pump is in auto mode
	IF NOT gCooling.cmd.manualMode THEN
		IF gStateMachine.status.state = STATE_DRIVE OR (inverterMaxTemp > gCooling.cmd.inverterTempStartPump) OR (motorMaxTemp > gCooling.cmd.motorTempStartPump) THEN
			gCooling.outputs.do_pump[1] := TRUE;
		ELSE
			gCooling.outputs.do_pump[1] := FALSE;
		END_IF;
	END_IF

	(* Convert analog temperature inputs to temperatures in degrees *)
	FOR i := 0 TO 1 DO
		(* Cooling System Temperature approximated via 4th order polynomium *)
		gCooling.data.coolingSysTemp[i] := EXPT(gCooling.inputs.ai_coolingTemp[i],2) + 0.004914 * gCooling.inputs.ai_coolingTemp[i] - 44.62;
	END_FOR

	// If cooling system is not in manual mode (its in automatic mode)
	IF NOT gCooling.cmd.manualMode THEN
		FOR i := 0 TO 1 DO
			//IF gCooling.outputs.do_pump[i] THEN
			//IF INT_TO_UINT(gCooling.inputs.im_pumpCurrent[i]) < pumpOffCurrent THEN
			// No current is being drawn
			//	gCooling.status.pumpState[i] := PUMP_STATE_NOT_CONNECTED;
			//ELSIF INT_TO_UINT(gCooling.inputs.im_pumpCurrent[i]) > pumpOffCurrent AND INT_TO_UINT(gCooling.inputs.im_pumpCurrent[i]) < pumpOnCurrent THEN
			// Not enough current is being drawn
			//	gCooling.status.pumpState[i] := PUMP_STATE_NO_WATER;
			//ELSE
			// Normal amount of current is being drawn
//			IF gStateMachine.status.state = STATE_DRIVE OR (inverterMaxTemp > gCooling.cmd.inverterTempStartPump) OR (motorMaxTemp > gCooling.cmd.motorTempStartPump) THEN
//				gCooling.status.pumpState[i] := PUMP_STATE_OK;
//				gCooling.outputs.do_pump[i] := TRUE;
//			ELSE
//				gCooling.status.pumpState[i] := PUMP_STATE_NO_WATER; // Just to turn off when not in tractive
//				gCooling.outputs.do_pump[i] := FALSE;
//			END_IF;
//
//			// Check if there is an error on the pump. If the pump state is not OK there is an error
//			gCooling.status.pumpError[i] := gCooling.status.pumpState[i] <> PUMP_STATE_OK;
//
//			// If there is an error turn OFF the pump. Otherwise keep it ON
//			gCooling.outputs.do_pump[i] := NOT gCooling.status.pumpError[i];
//
//			//END_IF

		END_FOR
	END_IF;

	// Enable fan when in STATE_DRIVE
	FOR i := 0 TO 1 DO
		gCooling.outputs.do_fan[i] := gStateMachine.status.state = STATE_DRIVE;
	END_FOR;

	// Evaluate if inverter or motors have high temperature errors
	gCooling.status.warningInverterHighTemp := MAX(gInverters.inverter[0].data.tempInverter, gInverters.inverter[1].data.tempInverter, gInverters.inverter[2].data.tempInverter, gInverters.inverter[3].data.tempInverter) > gCooling.cmd.inverterMaxTemp;
	gCooling.status.warningMotorHighTemp 	:= MAX(gInverters.inverter[0].data.tempMotor   , gInverters.inverter[1].data.tempMotor,    gInverters.inverter[2].data.tempMotor,    gInverters.inverter[3].data.tempMotor)    > gCooling.cmd.motorMaxTemp;

	// Evaluate if the cooling system is working properly.
	gCooling.status.ok := NOT gCooling.status.pumpError[0] AND NOT gCooling.status.pumpError[1];

	// Evaluate if the cooling system sees any temperature higher than allowed
	gCooling.status.warningHighTemperature := gCooling.status.warningInverterHighTemp OR gCooling.status.warningMotorHighTemp;
END_PROGRAM

PROGRAM _EXIT
	(* Insert code here *)

END_PROGRAM
```

### globalINS.var
```iecst
VAR
	gINS : gINS_typ;
END_VAR
```

### Types.typ
```iecst
(*Enumeration for Statemachine*)

TYPE
	enRECV_STEPS :
		(
		FRM_WAIT := 0, (*Defines the wait step*)
		FRM_OPEN, (*Defines Step for FRM_xopen() *)
		FRM_READ, (*Defines Step for FRM_read()*)
		FRM_COPY_RD_DATA, (*Defines Step for storing read data*)
		FRM_RBUF, (*Defines Step for FRM_rbuf()*)
		FRM_CLOSE, (*Defines Step for FRM_close()*)
		FRM_ERROR := 255 (*Defines Step for Errorhandling*)
		);
END_TYPE

(*Command data type*)

TYPE
	command_typ : 	STRUCT
		open_receive : BOOL; (*Open serial port and receive data*)
		close : BOOL; (*Close serial port*)
	END_STRUCT;
END_TYPE

(*Receiver type*)

TYPE
	Receiver_typ : 	STRUCT
		step : enRECV_STEPS; (*Step of the Statemachine*)
		Commands : command_typ; (*Commandinterface*)
		receive_data : STRING[80]; (*receive data*)
		FRM_xopen_0 : FRM_xopen; (*Functionblock FRM_xopen()*)
		xopenConfig : XOPENCONFIG; (*Configuration Type for FRM_xopen()*)
		FRM_read_0 : FRM_read; (*Functionblock FRM_read()*)
		FRM_rbuf_0 : FRM_rbuf; (*Functionblock FRM_rbuf()*)
		FRM_close_0 : FRM_close; (*Functionblock FRM_close()*)
	END_STRUCT;
END_TYPE
```

### Program Logical/Misc/DataLogging/DataLog (IEC)

#### DataLog.st - Init, cyclic, exit code
```iecst
PROGRAM _INIT

	RTInfo_0(enable := TRUE);
	initSetup;

END_PROGRAM

PROGRAM _CYCLIC
	// call actions
	// setup;
	setupFile;

	//detect if config.enable is changed then restart datalog
	FOR i:=0 TO DATALOG_MAX_MAPP_VARS DO
		IF this.okToRestart AND this.pvRegData[i].variable <> '' THEN
			IF this.pvRegData[i].address <> 0 AND this.pvRegData[i].datalength = 1 THEN
				pBool ACCESS this.pvRegData[i].address;
				IF pBool <> this.pvRegData[i].enable THEN
					this.state := 0; //restart
				END_IF
			END_IF
		ELSE EXIT;
		END_IF
	END_FOR

	//if file is changed then restart datalog
	FileInfo_0();
	IF this.okToRestart AND this.timestamp.old <> this.fileInfoSetting.modTime THEN
		this.state := 0; //restart
	END_IF

	CASE this.state OF
		0:	// wait for connected usb device
			IF gBrdkFileDev_0.description = 'all file devices are ready to use' THEN
				// finds the first available node
				FOR i := 1 TO BRDK_USB_MAX_DEVICES-1 DO
					IF gBrdkFileDev_0.availableDevices[i] <> '' THEN
						this.FileCreate_0.pDevice	:= ADR(gBrdkFileDev_0.availableDevices[i]);
						this.state := 5;
					END_IF
				END_FOR
			END_IF

		5: //create log folder
			this.okToRestart := FALSE;
			this.timestamp.old := this.fileInfoSetting.modTime;
			MpDataRecorder_0.Enable := FALSE;
			DirCreate_0.enable := TRUE;
			IF DirCreate_0.status = fiERR_DIR_ALREADY_EXIST THEN
				DirCreate_0.enable := FALSE;
				this.state := 10;
			END_IF
			DirCreate_0();

		10:
			MpRecipeRegPar_csv.Enable := TRUE;
			IF MpRecipeRegPar_csv.Active THEN
				this.state := 20;
			ELSIF MpRecipeRegPar_csv.Error THEN
				this.state := 65000;
			END_IF

		20:
			MpRecipeCsv_0.Enable := TRUE;
			IF MpRecipeCsv_0.Active THEN
				this.state := 30;
			ELSIF MpRecipeCsv_0.Error THEN
				this.state := 65000;
			END_IF

		30: //DatalogSettings.csv ok?
			IF FileInfo_0.status = ERR_OK THEN
				this.state := 40;
			ELSIF FileInfo_0.status = fiERR_FILE_NOT_FOUND THEN
				this.state := 300;
			ELSIF FileInfo_0.status = ERR_FUB_BUSY THEN
			ELSE
				this.state := 65000;
			END_IF

		40:
			MpRecipeCsv_0.Load := TRUE;
			IF MpRecipeCsv_0.CommandDone THEN
				MpRecipeCsv_0.Load := FALSE;
				this.state := 45;
			ELSIF MpRecipeCsv_0.Error THEN
				this.state := 65000;
			END_IF

		45:
			MpDataRecorder_0.Enable := TRUE;
			IF MpDataRecorder_0.Active THEN
				this.state := 50;
			ELSIF MpDataRecorder_0.Error THEN
				this.state := 65000;
			END_IF

		50://find logVar#logVarEnable and split it
			brsmemset(ADR(this.pvRegData), 0, SIZEOF(this.pvRegData));
			brsmemset(ADR(this.pvData), 0, SIZEOF(this.pvData));
			FOR i:=0 TO DATALOG_MAX_LOG_VARS DO
				IF gDataLogging.data.csvData[i] <> '' THEN
					this.strIdxPos := brdkStrSearch(ADR(gDataLogging.data.csvData[i]),ADR('#'));
					IF this.strIdxPos > 0 THEN //enable/disable variable found
						this.pvData[i].variable 	:= gDataLogging.data.csvData[i];
						this.pvData[i].enableVar 	:= gDataLogging.data.csvData[i];
						brdkStrSlice(ADR(this.pvData[i].variable), 0, this.strIdxPos);
						brdkStrSlice(ADR(this.pvData[i].enableVar), this.strIdxPos+1, SIZEOF(this.pvData[i].enableVar));
					ELSE
						this.pvData[i].variable := gDataLogging.data.csvData[i];
					END_IF
				ELSE EXIT;
				END_IF
			END_FOR
			this.state := 60;

		60://find and replace [x]. to [0..this.maxIdxVariableX]
			noOfPvVars := 0;
			FOR i:=0 TO DATALOG_MAX_LOG_VARS DO
				IF gDataLogging.data.csvData[i] <> '' THEN
					this.strIdxPos := brdkStrSearch(ADR(this.pvData[i].variable), ADR('[x]'));
				 	IF this.strIdxPos > 0 THEN
				 		FOR j:=0 TO this.maxIdxVariableX DO
							this.tmpStr := '[x]';
							brsitoa(j, ADR(this.idxStr));
							brdkStrReplace(ADR(this.tmpStr), ADR('x'), ADR(this.idxStr));
							this.pvRegData[noOfPvVars].variable 	:= this.pvData[i].variable;
							this.pvRegData[noOfPvVars].enableVar 	:= this.pvData[i].enableVar;
							brdkStrReplace(ADR(this.pvRegData[noOfPvVars].variable), ADR('[x]'), ADR(this.tmpStr));
							brdkStrReplace(ADR(this.pvRegData[noOfPvVars].enableVar), ADR('[x]'), ADR(this.tmpStr));
							PV_xgetadr(ADR(this.pvRegData[noOfPvVars].enableVar), ADR(this.pvRegData[noOfPvVars].address), ADR(this.pvRegData[noOfPvVars].datalength));
							noOfPvVars := noOfPvVars + 1;
						END_FOR
					ELSE
						this.pvRegData[noOfPvVars].variable 	:= this.pvData[i].variable;
						this.pvRegData[noOfPvVars].enableVar 	:= this.pvData[i].enableVar;
						PV_xgetadr(ADR(this.pvRegData[noOfPvVars].enableVar), ADR(this.pvRegData[noOfPvVars].address), ADR(this.pvRegData[noOfPvVars].datalength));
						noOfPvVars := noOfPvVars + 1;
				 	END_IF
				ELSE EXIT;
				END_IF
			END_FOR
			this.state := 65;

		65: //clear all reg pars before init again
			FOR i:=0 TO DATALOG_MAX_MAPP_VARS DO
				this.MpDataRegPar[i].Enable := FALSE;
			END_FOR
			this.state := 70;

		70: //registre pv's
			FOR i:=0 TO DATALOG_MAX_MAPP_VARS DO
				IF this.pvRegData[i].variable <> '' THEN
					this.MpDataRegPar[i].MpLink 		:= ADR(gDataRecorder);
					this.MpDataRegPar[i].Description 	:= ADR(this.pvRegData[i].variable);
					this.MpDataRegPar[i].PVName			:= ADR(this.pvRegData[i].variable);
					IF this.pvRegData[i].address <> 0 AND this.pvRegData[i].datalength = 1 THEN
						pBool ACCESS this.pvRegData[i].address;
						this.pvRegData[i].enable := pBool;
					ELSE
						this.pvRegData[i].enable := TRUE;
					END_IF
					this.MpDataRegPar[i].Enable	:= this.pvRegData[i].enable;
				ELSE EXIT;
				END_IF
			END_FOR
			this.okToRestart := TRUE;
			this.state := 80;

		80: //wait for system up and running
			IF this.systemReadyToLog THEN
				MpDataRecorder_0.Enable := TRUE;
				this.state := 85;
			END_IF

		85: //active
			IF MpDataRecorder_0.Active THEN
				this.TON_recordDelay.IN := TRUE;
				this.state := 90;
			ELSIF MpDataRecorder_0.Error THEN
				this.state := 65000;
			END_IF

		90: //delay before start recording
			IF this.TON_recordDelay.Q THEN
				this.TON_recordDelay.IN := FALSE;
				MpDataRecorder_0.Record := TRUE;
				this.state := 100;
			END_IF

		100: //ready
			gDataLogging.status.dataloggingActive := TRUE;
			IF gCreateLogFile THEN
				this.okToRestart := FALSE;
				MpDataRecorder_0.SnapShot := TRUE;
				this.state := 110;
			ELSIF NOT MpDataRecorder_0.Enable THEN // restart after download
				gCreateLogFile := FALSE;
				this.state := 0;
			ELSIF MpDataRecorder_0.Error THEN
				gCreateLogFile := FALSE;
				this.state := 65000;
			END_IF

			IF MpDataRecorder_0.Info.CurrentFileSize > 900 THEN
				this.state := 5;
			END_IF

		110: //waiting for datalog file created
			IF MpDataRecorder_0.SnapShotDone THEN
				MpDataRecorder_0.SnapShot 	:= FALSE;
				gCreateLogFile 				:= FALSE;
				this.state 					:= 100;
			ELSIF MpDataRecorder_0.Error THEN
				MpDataRecorder_0.ErrorReset	:= TRUE;
				MpDataRecorder_0.SnapShot 	:= FALSE;
				gCreateLogFile 				:= FALSE;
				this.state 					:= 65000;
			END_IF

		300: //create DatalogSettings.csv
			MpRecipeCsv_0.Save := TRUE;
			IF MpRecipeCsv_0.CommandDone THEN
				MpRecipeCsv_0.Save := FALSE;
				this.state := 0;
			ELSIF MpRecipeCsv_0.Error THEN
				this.state := 65000;
			END_IF

		65000://ERROR HANDLING = NONE :/
			this.TON_errorReset.IN	:= TRUE;
			IF this.TON_errorReset.Q THEN
				this.TON_errorReset.IN		:= FALSE;
				MpDataRecorder_0.Enable 	:= FALSE;
				MpRecipeRegPar_csv.Enable 	:= FALSE;
				MpRecipeCsv_0.Enable		:= FALSE;
				FileInfo_0.enable			:= FALSE;
				this.state					:= 0;
			END_IF

	END_CASE

	// Function Block Calls
	this.TON_errorReset(PT := T#10s);

	IF this.state <> 100 OR this.brdkUSBConnect_0.status <> BRDK_USB_STATUS_FB_READY THEN
		gDataLogging.status.dataloggingActive := FALSE;
	END_IF

	this.TON_recordDelay();
	IF MpDataRecorder_0.Active THEN
		FOR i:=0 TO DATALOG_MAX_MAPP_VARS DO
			this.MpDataRegPar[i]();
		END_FOR
	END_IF
	MpDataRecorderConfig_0();
	MpDataRecorder_0();
	MpRecipeRegPar_csv();
	MpRecipeCsv_0();
	this.brdkUSBConnect_0();

END_PROGRAM

PROGRAM _EXIT
	// Disable Mapp Function Blocks
	MpDataRecorder_0(Enable := FALSE);
	MpDataRecorderConfig_0(Enable := FALSE);
	MpRecipeCsv_0(Enable := FALSE);
	MpRecipeRegPar_csv(Enable := FALSE);
END_PROGRAM
```

#### setupFile.st
```iecst
ACTION setupFile:
	IF gBrdkFileDev_0.availableDevices[1] <> '' THEN
		MpRecipeRegPar_csv.MpLink 	:= ADR(gRecipeCsv);
		MpRecipeRegPar_csv.PVName 	:= ADR('DataLog:gDataLogging.inputs.csvData');
		MpRecipeRegPar_csv.Category	:= ADR('datalogSettings');

		MpRecipeCsv_0.MpLink 		:= ADR(gRecipeCsv);
		MpRecipeCsv_0.DeviceName 	:= ADR(gBrdkFileDev_0.availableDevices[1]);
		MpRecipeCsv_0.FileName 		:= ADR('log/DatalogSettings');
		MpRecipeCsv_0.Category		:= ADR('datalogSettings');

		MpDataRecorder_0.MpLink			:= ADR(gDataRecorder);
		MpDataRecorder_0.DeviceName		:= ADR(gBrdkFileDev_0.availableDevices[1]);
		MpDataRecorder_0.RecordMode 	:= mpDATA_RECORD_MODE_TIME;
		MpDataRecorder_0.SamplingTime	:= RTInfo_0.cycle_time / 1000; //micro to milli

		MpDataRecorderConfiguration.DecimalDigits	:= 3;
		MpDataRecorderConfiguration.BufferSize		:= 50000; //kB
		MpDataRecorderConfiguration.PowerFailSafe	:= FALSE;
		MpDataRecorderConfiguration.FileNamePattern	:= 'Datalog_%Y%m%d_%H%M%S.csv';
		MpDataRecorderConfiguration.DecimalMark		:= '.';
		MpDataRecorderConfiguration.AutoSave		:= FALSE;

		MpDataRecorderConfig_0.MpLink 				:= ADR(gDataRecorder);
		MpDataRecorderConfig_0.Configuration		:= ADR(MpDataRecorderConfiguration);
		MpDataRecorderConfig_0.Enable 				:= TRUE;

		FileInfo_0.pDevice			:= ADR(gBrdkFileDev_0.availableDevices[1]);
		FileInfo_0.pName			:= ADR('log/DatalogSettings.csv');
		FileInfo_0.pInfo			:= ADR(this.fileInfoSetting);
		FileInfo_0.enable			:= TRUE;

		DirCreate_0.pDevice			:= ADR(gBrdkFileDev_0.availableDevices[1]);
		DirCreate_0.pName			:= ADR('log');

		this.TON_recordDelay.PT 	:= T#10ms;
		this.maxIdxVariableX 		:= 0;
		this.systemReadyToLog 		:= TRUE;
	END_IF
END_ACTION
```

#### initSetup.st
```iecst
	//(* Writing the data to be datalogged *)
ACTION initSetup:

	// State
	gDataLogging.data.csvData[0] := 'gStateMachine.status.stateName';
	// Mission
	gDataLogging.data.csvData[1] := 'gStateMachine.status.mission';
	// Instruction
	gDataLogging.data.csvData[2] := 'gStateMachine.status.instruction';

	// ******* Dashboard information
	// State
	gDataLogging.data.csvData[3] := 'gDashboard.status.DashboardDisconnected';
	gDataLogging.data.csvData[4] := 'gDashboard.status.errorCode';
	// Buttons
	gDataLogging.data.csvData[5] := 'gDashboard.inputs.di_button1';
	gDataLogging.data.csvData[6] := 'gDashboard.inputs.di_button2';
	gDataLogging.data.csvData[7] := 'gDashboard.inputs.di_button3';
	gDataLogging.data.csvData[8] := 'gDashboard.inputs.di_button4';
	gDataLogging.data.csvData[9] := 'gDashboard.inputs.di_buttonSafety';
	gDataLogging.data.csvData[10] := 'gDashboard.inputs.di_buttonTractive';
	gDataLogging.data.csvData[11] := 'gDashboard.inputs.di_buttonDrive';

	// LED's
	gDataLogging.data.csvData[12] := 'gDashboard.outputs.do_ledAMS';
	gDataLogging.data.csvData[13] := 'gDashboard.outputs.do_ledIMD';
	gDataLogging.data.csvData[14] := 'gDashboard.outputs.do_ledLV';
	gDataLogging.data.csvData[15] := 'gDashboard.outputs.do_ledREADY';
	gDataLogging.data.csvData[16] := 'gDashboard.outputs.do_ledSC';
	gDataLogging.data.csvData[17] := 'gDashboard.outputs.do_ledTS_OFF';

END_ACTION
```

### globalDataLogging.var
```iecst
VAR
	gDataLogging : gDataLogging_typ;
END_VAR
VAR CONSTANT
	DATALOG_MAX_LOG_VARS : UINT := 300;
	DATALOG_MAX_MAPP_VARS : UINT := DATALOG_MAX_LOG_VARS;
END_VAR
VAR
	gCreateLogFile : BOOL;
END_VAR
```

### Program Logical/Misc/DataLogging/NewLogging (IEC)

#### Main.st - Init, cyclic, exit code
```iecst
PROGRAM _INIT
	this ACCESS ADR(local);
	(* Insert code here *)
	mpDataRecorder_0.MpLink 		:= ADR(gDataRecorderNew);
	mpDataRecorder_0.Enable 		:= FALSE;
	mpDataRecorder_0.SamplingTime := T#20ms; //[ms]
	mpDataRecorder_0.RecordMode	:= mpDATA_RECORD_MODE_TIME;

	mpDataRecorderConfig_0.MpLink := ADR(gDataRecorderNew);
	mpDataRecorderConfig_0.Configuration := ADR(mpDataRecorderConfigPar);
	mpDataRecorderConfig_0.Enable := TRUE;

	setupLog;
END_PROGRAM

PROGRAM _CYCLIC
	this ACCESS ADR(local);
	(* Insert code here *)

	CASE this.state OF
		0:
			this.stateinfo := 'Waiting for filedevices';
			mpDataRecorder_0.Record := FALSE;

			IF gBrdkFileDev_0.ready  THEN
				this.state := 1;
			END_IF

		1: // Activate config load = TRUE
			mpDataRecorderConfig_0.Load := TRUE;

			IF mpDataRecorderConfig_0.CommandDone THEN
				mpDataRecorderConfig_0.Load := FALSE;
				this.state := 10;
			END_IF

		5: //Wait for activate logging command

		10:
			this.stateinfo := 'Setting up Data Recorder';
			mpDataRecorder_0.DeviceName := ADR('LOG');
			mpDataRecorder_0.Enable	:= TRUE;

			IF mpDataRecorder_0.Error THEN
				this.state := 9999;
			ELSIF mpDataRecorder_0.Active THEN
				IF mpDataRecorder_0.Info.RegisteredPVCount = NUM_LOG_VAR THEN
					this.state := 20;
				ELSE
					this.state := 900;
				END_IF;
			END_IF;

		20:
			this.stateinfo := 'Waiting for Enabling in LiveView';
			IF (this.activateLogging) THEN
				mpDataRecorder_0.Record := TRUE;
			ELSIF this.setFilename THEN
				this.state := 200;
				this.setFilename := FALSE;
			END_IF

			IF mpDataRecorder_0.Recording THEN
				this.state := 100;
			ELSIF mpDataRecorder_0.Error THEN
				this.state := 9999;
			END_IF;

		100:
			this.stateinfo := 'Data is being recorded';

			IF NOT (this.activateLogging) THEN

				mpDataRecorder_0.Record := FALSE;
				this.state := 0;
			END_IF;

			IF mpDataRecorder_0.Error THEN
				this.state := 9999;
			END_IF
		200:
			// change name
			// Set save = true
			IF this.newFilename <> '' THEN
				mpDataRecorderConfigPar.FileNamePattern := this.newFilename;
				this.newFilename := '';
			END_IF;

			mpDataRecorderConfig_0.Save := TRUE;

			IF mpDataRecorderConfig_0.CommandDone THEN
				mpDataRecorderConfig_0.Save := FALSE;
				this.state := 20;
			END_IF

		900:
			this.stateinfo := 'Re-Enable mpdatalog';
			mpDataRecorder_0.Record := FALSE;
			this.state := 10;

		9999:
			this.stateinfo := 'ERROR';

			mpDataRecorder_0.Record := FALSE;
			mpDataRecorder_0.ErrorReset := TRUE;

			IF NOT mpDataRecorder_0.Error THEN
				mpDataRecorder_0.ErrorReset := FALSE;
	  			this.state := 0;
			END_IF;

	END_CASE

	this.loggingActive := mpDataRecorder_0.Recording;
	this.filename := mpDataRecorder_0.Info.CurrentFileName;

	mpDataRecorderConfig_0();
	mpDataRecorder_0();

	FOR i := 0 TO MAX_LOG_VAR DO
		IF mpDataRegPar_0[i].Active THEN
			mpDataRegPar_0[i]();
		ELSE
			EXIT;
		END_IF;
	END_FOR;

END_PROGRAM

PROGRAM _EXIT
	(* Insert code here *)
	mpDataRecorder_0(Enable := FALSE);

END_PROGRAM
```

#### Types.typ - Local data types
```iecst
TYPE
	local_typ : 	STRUCT
		stateinfo : STRING[50];
		state : UINT;
		activateLogging : BOOL;
		loggingActive : BOOL := FALSE;
		newFilename : STRING[50] := 'Datalog_%m_%d_%H_%M.csv';
		filename : STRING[50];
		activateLoggingArduino : BOOL := FALSE;
		setFilename : BOOL := FALSE;
	END_STRUCT;
END_TYPE
```

#### Variables.var - Local variables
```iecst
VAR
	mpDataRecorder_0 : MpDataRecorder;
	mpDataRecorderConfigPar : MpDataRecorderConfigType;
	mpDataRecorderConfig_0 : MpDataRecorderConfig;
	mpDataRegPar_0 : ARRAY[0..MAX_LOG_VAR] OF MpDataRegPar;
	local : local_typ;
	this : REFERENCE TO local_typ;
END_VAR
VAR CONSTANT
	MAX_LOG_VAR : USINT := 38;
END_VAR
VAR
	i : INT;
	loggingNames : ARRAY[0..MAX_LOG_VAR] OF STRING[80];
END_VAR
VAR CONSTANT
	NUM_LOG_VAR : USINT := MAX_LOG_VAR +1;
END_VAR
```

#### setupLog.st
```iecst
ACTION setupLog:

	//Variables to log
	loggingNames[0] := 'gStateMachine.status.state';
	loggingNames[1] := 'SENSORS:suspension.status.travelFL';
	loggingNames[2] := 'SENSORS:suspension.status.travelFR';
	loggingNames[3] := 'gSteeringAngle.data.angleDegrees';
	loggingNames[4] := 'gBraking.data.pressurePercentageRear';
	loggingNames[5] := 'gTorqueSensor.status.torquePercentage';
	loggingNames[6] := 'gInverters.inverter[0].data.actualVelocityKmh';
	loggingNames[7] := 'gInverters.inverter[1].data.actualVelocityKmh';
	loggingNames[8] := 'gInverters.inverter[2].data.actualVelocityKmh';
	loggingNames[9] := 'gInverters.inverter[3].data.actualVelocityKmh';
	loggingNames[10] := 'gInverters.inverter[0].outputs.com_torqueLimitPos';
	loggingNames[11] := 'gInverters.inverter[1].outputs.com_torqueLimitPos';
	loggingNames[12] := 'gInverters.inverter[2].outputs.com_torqueLimitPos';
	loggingNames[13] := 'gInverters.inverter[3].outputs.com_torqueLimitPos';
	loggingNames[14] := 'gInverters.inverter[0].data.torqueCurrent';
	loggingNames[15] := 'gInverters.inverter[1].data.torqueCurrent';
	loggingNames[16] := 'gInverters.inverter[2].data.torqueCurrent';
	loggingNames[17] := 'gInverters.inverter[3].data.torqueCurrent';
	loggingNames[18] := 'gInverters.inverter[0].data.torqueMagnitizingCurrent';
	loggingNames[19] := 'gInverters.inverter[1].data.torqueMagnitizingCurrent';
	loggingNames[20] := 'gInverters.inverter[2].data.torqueMagnitizingCurrent';
	loggingNames[21] := 'gInverters.inverter[3].data.torqueMagnitizingCurrent';
	loggingNames[22] := 'gInverters.inverter[0].data.tempInverter';
	loggingNames[23] := 'gInverters.inverter[1].data.tempInverter';
	loggingNames[24] := 'gInverters.inverter[2].data.tempInverter';
	loggingNames[25] := 'gInverters.inverter[3].data.tempInverter';
	loggingNames[26] := 'gInverters.inverter[0].data.tempMotor';
	loggingNames[27] := 'gInverters.inverter[1].data.tempMotor';
	loggingNames[28] := 'gInverters.inverter[2].data.tempMotor';
	loggingNames[29] := 'gInverters.inverter[3].data.tempMotor';
	loggingNames[30] := 'gAMS.data.cellTempMax';
	loggingNames[31] := 'gORION.data.packVoltage';
	loggingNames[32] := 'gORION.data.outputCurrent';
	loggingNames[33] := 'gTorqueSensor.data.torque1Percent';
	loggingNames[34] := 'gTorqueSensor.data.torque2Percent';
	loggingNames[35] := 'gORION.data.packPower';
	loggingNames[36] := 'SENSORS:accelerometer.input.x_direction';
	loggingNames[37] := 'SENSORS:accelerometer.input.y_direction';
	loggingNames[38] := 'SENSORS:accelerometer.input.z_direction';

	FOR i := 0 TO MAX_LOG_VAR DO
		mpDataRegPar_0[i].MpLink := ADR(gDataRecorderNew);
		mpDataRegPar_0[i].PVName := ADR(loggingNames[i]);
		mpDataRegPar_0[i].Enable := TRUE;
		mpDataRegPar_0[i]();
	END_FOR

END_ACTION
```

- Visualisation Logical/mappView (not shown)

### Program Logical/File/file (IEC)

#### Types.typ
```iecst
TYPE
	local_typ : 	STRUCT
		brdkFileDevUsb : brdkFileDeviceHandler;
		brdkFileDev : brdkFileDeviceHandler;
		lastFileName : STRING[255];
		brdkFileRead : brdkFileRead;
		fileName : STRING[255];
		fileType : STRING[5];
		delayTon : TON;
		setIdx : BOOL;
		stateInfo : STRING[40];
		state : UINT;
	END_STRUCT;
END_TYPE
```

#### Variables.var
```iecst
VAR
	this : local_typ;
END_VAR
VAR CONSTANT
	FILES_LIST_SIZE : USINT := 13; (*Number of files to be displayed on one page of the list in the HMI application*)
END_VAR
```

#### Main.st
```iecst
PROGRAM _INIT
	(* Insert code here *)
	gBrdkFileDev_0.enable := FALSE;
	gBrdkFileDev_0.setup.plcDrive := F_DRIVE;
	gBrdkFileDev_0.setup.usbOverrule := TRUE;
	gBrdkFileDev_0.simulation.pcRootFolder := 'Vikings';
	gBrdkFileDev_0.simulation.pcHDDrive := C_DRIVE;
	gBrdkFileDev_0.simulation.pcUSBDrive := D_DRIVE;

	gBrdkFileDev_0.setup.fileDevices[0].name 		:= 'LOG';
	gBrdkFileDev_0.setup.fileDevices[0].path 		:= 'x90log\log';
	gBrdkFileDev_0.setup.fileDevices[1].name 		:= 'TEMP';
	gBrdkFileDev_0.setup.fileDevices[1].path 		:= 'temp';

	// gBrdkFileDev_0.setup.fileDevices[0].useUSB		:= TRUE;

	this.delayTon.PT := T#2s;
	this.delayTon.IN := FALSE;

	this.state := 0;

	gBrdkFileDev_0();
END_PROGRAM

PROGRAM _CYCLIC

	CASE this.state OF
		0:
			this.stateInfo := 'Waiting for File Devices to be ready';
			gBrdkFileDev_0.enable := TRUE;
			IF gBrdkFileDev_0.ready THEN
	  			this.state := 100;
			END_IF;

			IF gBrdkFileDev_0.status <> 0 THEN
				this.state := 9999;
			END_IF;
		100:
			this.stateInfo := 'All file devices are ready';

			IF gBrdkFileDev_0.status <> 0 THEN
				this.state := 9999;
			END_IF;
		9999:
			this.stateInfo := 'error occured';
			// Flicking the enable input of File Dev handler
			IF this.delayTon.Q THEN
				this.delayTon.IN := FALSE;
				gBrdkFileDev_0.enable := NOT gBrdkFileDev_0.enable;
			ELSE
				this.delayTon.IN := TRUE;
			END_IF;

			IF gBrdkFileDev_0.ready THEN
	  			this.state := 100;
			END_IF;

	END_CASE;

	// Create file devices
	gBrdkFileDev_0();

	this.delayTon();
END_PROGRAM

PROGRAM _EXIT
	(* Insert code here *)
	 gBrdkFileDev_0(enable := FALSE);
END_PROGRAM
```

### gFile.typ
```iecst
TYPE
	gFile_input_typ : 	STRUCT
		refresh : BOOL;
	END_STRUCT;
	gFile_output_typ : 	STRUCT
		fileDevice : STRING[10];
		ready : BOOL;
	END_STRUCT;
	gFile_typ : 	STRUCT
		output : gFile_output_typ;
		input : gFile_input_typ;
	END_STRUCT;
END_TYPE
```

### gFile.var
```iecst
VAR
	gBrdkFileDev_0 : brdkFileDeviceHandler;
	gFile : gFile_typ;
END_VAR
```

### Program Logical/Inverters/CAN/CAN

#### Types.typ
```iecst
TYPE
	bus_typ : 	STRUCT
		ArCanSetBaudrate_0 : ArCanSetBaudrate;
		ArCanSend_0 : ArCanSend;
		ArCanReceive_0 : ArCanReceive;
		sendMessages : UDINT;
		receivedMessages : UDINT;
		deviceName : STRING[127];
		TON_detectTimer : ARRAY[0..1]OF TON;
		TON_sendTimer : TON;
		communicationState : CAN_STATES;
	END_STRUCT;
END_TYPE
```

#### Variables.var
```iecst
VAR
	k : USINT;
	inverterId : USINT;
	bus : ARRAY[0..1] OF bus_typ;
END_VAR
VAR CONSTANT
	MAX_SEND_MESSAGES_1 : USINT := 3;
	MAX_SEND_MESSAGES_0 : USINT := 3;
END_VAR
VAR
	i : USINT;
	j : USINT;
	RX_CAN_ID_BASE : UDINT;
	TX_CAN_ID_BASE : UDINT;
END_VAR
```

#### Main.st
```iecst
PROGRAM _INIT
	(* Devices *)
	bus[0].deviceName := 'IF7';
	bus[1].deviceName := 'IF8';

	FOR i := 0 TO 1 DO
		(* Bus *)
		bus[i].ArCanSetBaudrate_0.Baudrate 	:= 500000;
		(* Transmit *)
		bus[i].ArCanSend_0.Frame.Format 	:= arCAN_11BIT;

		(* Receive *)
		bus[i].ArCanReceive_0.Format 		:= arCAN_11BIT;
		bus[i].ArCanReceive_0.QueueSize		:= 100;
		bus[i].ArCanReceive_0.IDMask		:= arCAN_RECEIVE_ALL;

		bus[i].communicationState := S_INIT;

		(* Set timeout for timers and start them*)
		FOR j := 0 TO 1 DO
			bus[i].TON_detectTimer[j].PT := T#100ms;
			bus[i].TON_detectTimer[j].IN := TRUE;
		END_FOR

	END_FOR;

	RX_CAN_ID_BASE := 16#200;
	TX_CAN_ID_BASE := 16#100;

	// TEMP
	gInverters.status.torqueBasedThrottle := TRUE;
	//bus[0].communicationState := S_IDLE;

END_PROGRAM

PROGRAM _CYCLIC
	FOR i := 0 TO 1 DO
		Bus;
	END_FOR;
END_PROGRAM

PROGRAM _EXIT

END_PROGRAM
```

#### disconnectionDetecton.st
```iecst
ACTION serviceDisconnectionDetection:

	(* Check timeouts for inverters *)
	FOR j := 0 TO 1 DO
		bus[i].TON_detectTimer[j]();
		(* If timeout has occurred*)
		IF bus[i].TON_detectTimer[j].Q THEN
			(* Report error*)
			gInverters.inverter[(i*2)+j].status.inverterDisconnected := TRUE;
		ELSE
			(* Reset error *)
			gInverters.inverter[(i*2)+j].status.inverterDisconnected := FALSE;
		END_IF
	END_FOR
END_ACTION

ACTION updateDisconnectionDetection:

	IF inverterId = 0 OR inverterId = 2 THEN
		// Inverter 0 and 2 have index 0 in the detectTimer array
		j := 0;
	ELSE
		// Inverter 1 and 3 have index 1 in the detectTimer array
		j := 1;
	END_IF;

	// Reset timer and update it
	bus[i].TON_detectTimer[j].IN := FALSE;
	bus[i].TON_detectTimer[j]();

END_ACTION
```

#### Program Logical/Inverters/CAN/CAN/Send

##### encodeAndSendMessage.st
```iecst
ACTION encodeAndSendMessage:
	(* Write data *)
	(* Booleans *)
	bus[i].ArCanSend_0.Frame.Data[1].0 := gInverters.inverter[j].outputs.com_interverOn;
	bus[i].ArCanSend_0.Frame.Data[1].1 := gInverters.inverter[j].outputs.com_dcOn;
	bus[i].ArCanSend_0.Frame.Data[1].2 := gInverters.inverter[j].outputs.com_enable;
	bus[i].ArCanSend_0.Frame.Data[1].3 := gInverters.inverter[j].outputs.com_errorReset;

	(* Integers *)
	IF gInverters.status.torqueBasedThrottle THEN // If throttle should be torque based, set velocity to max velocity
		IF gInverters.inverter[j].outputs.com_targetTorque > 0 THEN
			gInverters.inverter[j].outputs.com_targetTorque := gInverters.inverter[j].outputs.com_targetVelocity ; // Max RPM of motor
		ELSE
			gInverters.inverter[j].outputs.com_targetTorque := 0;
		END_IF;
	END_IF
	memcpy(ADR(bus[i].ArCanSend_0.Frame.Data[2]),ADR(gInverters.inverter[j].outputs.com_targetTorque), 2); // ACtually velocity setpoint [rpm]

	IF gInverters.inverter[j].outputs.com_torqueLimitPos < 0 THEN
	  gInverters.inverter[j].outputs.com_torqueLimitPos := 0;
	END_IF;
	memcpy(ADR(bus[i].ArCanSend_0.Frame.Data[4]),ADR(gInverters.inverter[j].outputs.com_torqueLimitPos), 2);
	memcpy(ADR(bus[i].ArCanSend_0.Frame.Data[6]),ADR(gInverters.inverter[j].outputs.com_torqueLimitNeg), 2);

	IF NOT gIsSimulation THEN

		(* Set DLC *)
		bus[i].ArCanSend_0.Frame.DataLength 	:= 8;

		(* Send message *)
		bus[i].ArCanSend_0(SendFrame := TRUE);
		bus[i].ArCanSend_0(SendFrame := FALSE);
	END_IF;
END_ACTION
```

### Program Logical/Inverters/Control/Control (IEC)

#### powerLimiter.st
```iecst
ACTION powerLimiterInit:
	// Initialize the controller values
	gInverters.data.powerLimitKW := 50;
	gInverters.data.powerLimitMargin := 0.9;

	//control.PL.enable 		 := gInverters.cmd.enablePowerLimiter;
	//control.PL.MAX_POWER	 := gInverters.data.powerLimitKW; // [kW]
	//FOR i := 0 TO INVERTER_COUNT DO
	//	control.PL.I_GAIN[i] := 0;
	//	control.PL.P_GAIN[i] := 0;
	//END_FOR;
	constant.NOMINAL_TORQUE := 9.8; // [Nm]
	constant.MAX_TORQUE 	:= 21; // [Nm]
END_ACTION

ACTION powerLimiterCyclic:
	// Service the controller
	gInverters.data.MaxSpeedRPM :=  MAX(gInverters.inverter[0].data.actualVelocity, gInverters.inverter[1].data.actualVelocity, gInverters.inverter[2].data.actualVelocity, gInverters.inverter[3].data.actualVelocity, 1);
	MaxSpeedRADS := (gInverters.data.MaxSpeedRPM*2*constant.PI)/60;
	torqueLimitNM := ((MIN(gInverters.data.powerLimitKW,gORION.data.DCL_KW) /4)*1000)/MaxSpeedRADS * gInverters.data.powerLimitMargin; // 0.9 is equvivalent to 10% margin of limit
	gInverters.inverter[i].outputs.com_torqueLimitPos 	:= DINT_TO_INT(LIMIT(0,REAL_TO_DINT((torqueLimitNM/constant.NOMINAL_TORQUE)*1000), 32767)); // Is sent as 0.1% of nominel torque

	//control.PL.enable 				:= gInverters.cmd.enablePowerLimiter; // This might needed to be turned on?
	//control.PL.act_power			:= gShunt.data.actPowerKW;
	//control.PL.lowest_cell_voltage 	:= MIN(gAMS.data.cellVoltageMin[0], gAMS.data.cellVoltageMin[1], gAMS.data.cellVoltageMin[2], gAMS.data.cellVoltageMin[3], gAMS.data.cellVoltageMin[4]);
	//control.PL();
END_ACTION

ACTION powerLimiterCyclicIndividual:
	// Service the controller
	ActualSpeedRADS := (MAX(gInverters.inverter[i].data.actualVelocity, 1)*2*constant.PI)/60;
	torqueLimitNM := (gInverters.data.powerLimitKwInverter[i]*1000)/ActualSpeedRADS * gInverters.data.powerLimitMargin; // 0.9 is equvivalent to 10% margin of limit
	gInverters.inverter[i].outputs.com_torqueLimitPos 	:= DINT_TO_INT(LIMIT(0,REAL_TO_DINT((torqueLimitNM/constant.NOMINAL_TORQUE)*1000), 32767)); // Is sent as 0.1% of nominel torque

	//control.PL.enable 				:= gInverters.cmd.enablePowerLimiter; // This might needed to be turned on?
	//control.PL.act_power			:= gShunt.data.actPowerKW;
	//control.PL.lowest_cell_voltage 	:= MIN(gAMS.data.cellVoltageMin[0], gAMS.data.cellVoltageMin[1], gAMS.data.cellVoltageMin[2], gAMS.data.cellVoltageMin[3], gAMS.data.cellVoltageMin[4]);
	//control.PL();
END_ACTION
```

#### regenerativeBraking.st
```iecst
ACTION regenerativeBrakingInit:
	// Initialize the controller values
	control.RB.IDLE_MOTOR_TORQUE := 0.3; //[%/100]. 0.3 = 30%
END_ACTION

ACTION regenerativeBrakingCyclic:
	// Service the controller

//	control.RB.enable 		 	:= gInverters.cmd.enableRegenerativeBraking;
//	control.RB.brake_pressure	:= gBraking.data.pressurePercentage;
//	control.RB();
END_ACTION
```

#### convertToKmh.st
```iecst
ACTION convertToKmh:
	constant.GEAR_RATIO	  := 11.0118;
	constant.WHEEL_RADIUS := 0.195;
	constant.PI 		  := 3.141592;

	FOR i := 0 TO INVERTER_COUNT DO
		// Convert from RPM to KMH
		// Speed in km/h								=  (             Number of wheel rotations               		) * (       Wheel distance traveled	      ) * (m/min to km/h)
		gInverters.inverter[i].data.actualVelocityKmh := (gInverters.inverter[i].data.actualVelocity / constant.GEAR_RATIO) * (constant.WHEEL_RADIUS * 2 * constant.PI) * 0.06;
	END_FOR;

END_ACTION
```

#### history.st
```iecst
ACTION history:
	// Power history
//	TON_history.PT := T#10ms;
//	TON_history.IN := TRUE;
//	IF TON_history.Q THEN
//		FOR i := 999 TO 1 BY -1 DO
//			FOR j := 0 TO 3 DO
//				gInverter[j].data.history.actualVelocityKmh[i] 		 := gInverter[j].data.history.actualVelocityKmh[i-1];
//				gInverter[j].data.history.com_targetTorque[i] 		 := gInverter[j].data.history.com_targetTorque[i-1];
//				gInverter[j].data.history.deratingTotalPercentage[i] := gInverter[j].data.history.deratingTotalPercentage[i-1];
//				gInverter[j].data.history.steeringAngle[i] 			 := gInverter[j].data.history.steeringAngle[i-1];
//				gInverter[j].data.history.torqueMax[i] 				 := gInverter[j].data.history.torqueMax[i-1];
//				gInverter[j].data.history.torquePercentage[i] 		 := gInverter[j].data.history.torquePercentage[i-1];
//			END_FOR;
//		END_FOR;
//		FOR j := 0 TO 3 DO
//			gInverter[j].data.history.actualVelocityKmh[i] 		 := gInverter[j].data.actualVelocityKmh;
//			gInverter[j].data.history.com_targetTorque[i] 		 := gInverter[j].outputs.com_targetTorque;
//			gInverter[j].data.history.deratingTotalPercentage[i] := gInverter[j].status.deratingTotalPercent;
//			gInverter[j].data.history.steeringAngle[i] 			 := gSteeringAngle.data.angleDegrees;
//			gInverter[j].data.history.torqueMax[i] 				 := gInverters.data.torqueLimitNm;
//			gInverter[j].data.history.torquePercentage[i] 		 := gTorqueSensor.status.torquePercentage;
//		END_FOR;
//		TON_history.IN := FALSE;
//	END_IF;
//	TON_history();
END_ACTION
```

### Program Logical/Inverters/Inv_statemachine/Inv_statemachine (IEC)

#### hmiAction.st
```iecst
(* Convert values to show on liveview *)
ACTION hmiAction:
	(* Calculate correct values *)
	FOR i := 0 TO INVERTER_COUNT DO

		gInverters.inverter[i].data.tempIGBT 					:= gInverters.inverter[i].inputs.com_tempIGBT 	/ 10.00;
		gInverters.inverter[i].data.tempInverter 				:= gInverters.inverter[i].inputs.com_tempInverter / 10.00;
		gInverters.inverter[i].data.tempMotor 				:= gInverters.inverter[i].inputs.com_tempMotor 	/ 10.00;

		gInverters.inverter[i].data.actualVelocity 			:= gInverters.inverter[i].inputs.com_actualVelocity;
		gInverters.inverter[i].data.torqueCurrent 			:= (gInverters.inverter[i].inputs.com_torqueCurrent*CONVERTER_PEAK_CURRENT)	  /16384.00;
		gInverters.inverter[i].data.torqueMagnitizingCurrent 	:= (gInverters.inverter[i].inputs.com_magnetizingCurrent*CONVERTER_PEAK_CURRENT)/16384.00;
	END_FOR;

END_ACTION
```

### Program Logical/Inverters/Simulation/Simulation (IEC)

#### Variables.var
```iecst
VAR
	i : UINT;
END_VAR
VAR CONSTANT
	INVERTER_COUNT : USINT := 3;
END_VAR
```

Listed in the project but not available here: Logical/Global.typ, Logical/Libraries/brdkUSB/brdkUSB.typ, Logical/Libraries/brdkUSB/brdkUSB.var, Logical/Libraries/brdkUSB/brdkUSB.fun, Logical/Libraries/brdkFile/brdkFileCreateSubFolders.c, Logical/Libraries/brdkFile/brdkFile_func.h, Logical/globalEventLog.typ, Logical/globalEventLog.var, Logical/SM/StateMachine/functions/eventLog/logEvent.st, Logical/SM/StateMachine/functions/eventLog/logEvent.st, Logical/AMS_and_Shunt/globalAMS.var, Logical/AMS_and_Shunt/globalORION.typ, Logical/AMS_and_Shunt/globalShunt.typ, Logical/Dashboard/Dashboard/ledControl/ledAMS.st, Logical/Dashboard/Dashboard/ledControl/ledDV.st, Logical/Dashboard/Dashboard/ledControl/ledEBS.st, Logical/Dashboard/Dashboard/ledControl/ledIMD.st, Logical/Dashboard/Dashboard/ledControl/ledLV.st, Logical/Dashboard/Dashboard/ledControl/ledREADY.st, Logical/Dashboard/Dashboard/ledControl/ledSC.st, Logical/Sensors/globalSteeringAngle.typ, Logical/Sensors/globalSteeringAngle.var, Logical/Sensors/globalTorqueSensor.typ, Logical/Sensors/globalLowVoltageBattery.typ, Logical/Sensors/globalLowVoltageBattery.var, Logical/Sensors/Sensors/LowVoltageBattery, Logical/SensorNet/globalSensorNet/Types.typ, Logical/Misc/DataLogging/sampleST, Logical/Misc/DataLogging/DataLog/Types.typ, Logical/Misc/DataLogging/DataLog/Variables.var, Logical/Misc/DataLogging/DataLog/setup.st, Logical/Misc/DataLogging/globalDataLogging.typ, Logical/Inverters/globalInverters.typ, Logical/Inverters/globalInverters.var, Logical/Inverters/CAN/CAN/Receive/Receive_Bus.st, Logical/Inverters/CAN/CAN/Receive/Messages, Logical/Inverters/Control/Control/Main.st, Logical/Inverters/Control/Control/Types.typ, Logical/Inverters/Control/Control/Variables.var, Logical/Inverters/Control/Control/Mics/torqueOff.st, Logical/Inverters/Control/Control/Mics/frontRearDistribution.st, Logical/Inverters/Control/Control/Mics/accelerationMeasurement.st, Logical/Inverters/Inv_statemachine/Inv_statemachine/Main.st, Logical/Inverters/Inv_statemachine/Inv_statemachine/Types.typ, Logical/Inverters/Inv_statemachine/Inv_statemachine/Variables.var, Logical/Inverters/Inv_statemachine/Inv_statemachine/errorTimeout.st, Logical/Inverters/Inv_statemachine/Inv_statemachine/mission.st, Logical/SM/StateMachine/functions/eventLog/logEvent.st
